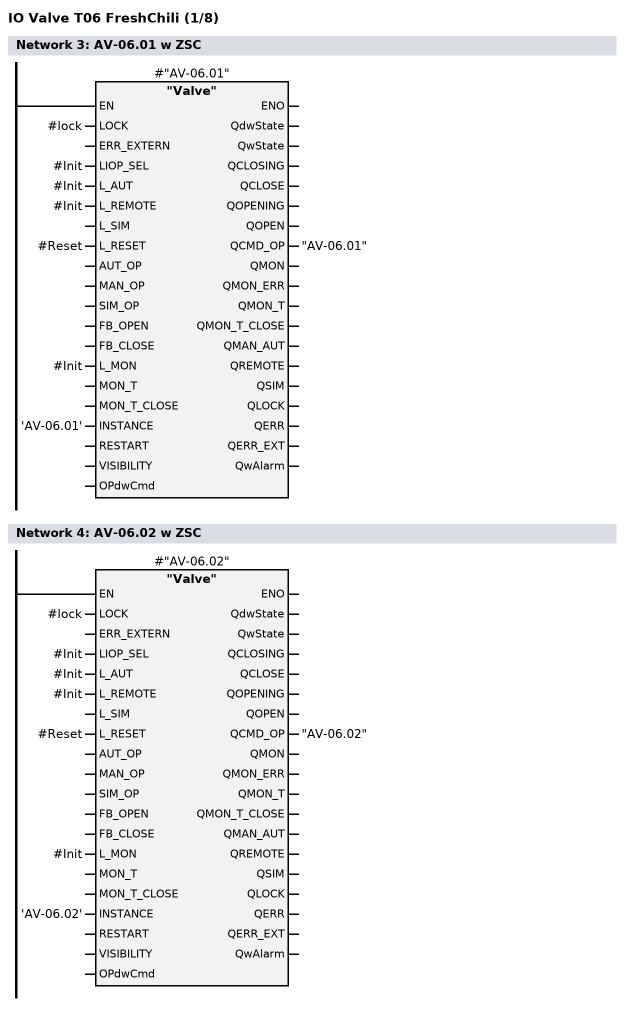
   RUNG wire#powerrail
      #"AV-06.01"(LOCK := #lock, ERR_EXTERN :=, LIOP_SEL := #Init, L_AUT := #Init, L_REMOTE := #Init, L_SIM :=, L_RESET := #Reset, AUT_OP :=, MAN_OP :=, SIM_OP :=, FB_OPEN :=, FB_CLOSE :=, L_MON := #Init, MON_T :=, MON_T_CLOSE :=, INSTANCE := 'AV-06.01', RESTART :=, VISIBILITY :=, OPdwCmd :=, QdwState =>, QwState =>, QCLOSING =>, QCLOSE =>, QOPENING =>, QOPEN =>, QCMD_OP => "AV-06.01", QMON =>, QMON_ERR =>, QMON_T =>, QMON_T_CLOSE =>, QMAN_AUT =>, QREMOTE =>, QSIM =>, QLOCK =>, QERR =>, QERR_EXT =>, QwAlarm =>)
   END_RUNG
   // the same network as SCL:
   #"AV-06.01"(LOCK := #lock,   // "Valve"
               LIOP_SEL := #Init,
               L_AUT := #Init,
               L_REMOTE := #Init,
               L_RESET := #Reset,
               L_MON := #Init,
               INSTANCE := 'AV-06.01',
               QCMD_OP => "AV-06.01");
END_REGION

REGION Network 4: AV-06.02 w ZSC
   RUNG wire#powerrail
      #"AV-06.02"(LOCK := #lock, ERR_EXTERN :=, LIOP_SEL := #Init, L_AUT := #Init, L_REMOTE := #Init, L_SIM :=, L_RESET := #Reset, AUT_OP :=, MAN_OP :=, SIM_OP :=, FB_OPEN :=, FB_CLOSE :=, L_MON := #Init, MON_T :=, MON_T_CLOSE :=, INSTANCE := 'AV-06.02', RESTART :=, VISIBILITY :=, OPdwCmd :=, QdwState =>, QwState =>, QCLOSING =>, QCLOSE =>, QOPENING =>, QOPEN =>, QCMD_OP => "AV-06.02", QMON =>, QMON_ERR =>, QMON_T =>, QMON_T_CLOSE =>, QMAN_AUT =>, QREMOTE =>, QSIM =>, QLOCK =>, QERR =>, QERR_EXT =>, QwAlarm =>)
   END_RUNG
   // the same network as SCL:
   #"AV-06.02"(LOCK := #lock,   // "Valve"
               LIOP_SEL := #Init,
               L_AUT := #Init,
               L_REMOTE := #Init,
               L_RESET := #Reset,
               L_MON := #Init,
               INSTANCE := 'AV-06.02',
               QCMD_OP => "AV-06.02");
END_REGION

REGION Network 5: AV-06.03 w ZSC
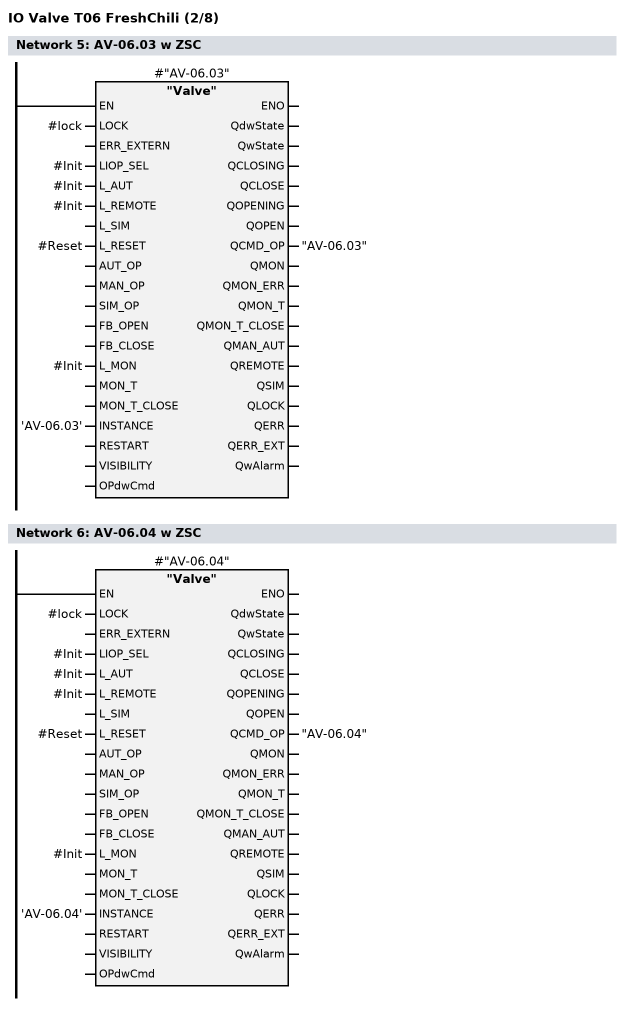
   RUNG wire#powerrail
      #"AV-06.03"(LOCK := #lock, ERR_EXTERN :=, LIOP_SEL := #Init, L_AUT := #Init, L_REMOTE := #Init, L_SIM :=, L_RESET := #Reset, AUT_OP :=, MAN_OP :=, SIM_OP :=, FB_OPEN :=, FB_CLOSE :=, L_MON := #Init, MON_T :=, MON_T_CLOSE :=, INSTANCE := 'AV-06.03', RESTART :=, VISIBILITY :=, OPdwCmd :=, QdwState =>, QwState =>, QCLOSING =>, QCLOSE =>, QOPENING =>, QOPEN =>, QCMD_OP => "AV-06.03", QMON =>, QMON_ERR =>, QMON_T =>, QMON_T_CLOSE =>, QMAN_AUT =>, QREMOTE =>, QSIM =>, QLOCK =>, QERR =>, QERR_EXT =>, QwAlarm =>)
   END_RUNG
   // the same network as SCL:
   #"AV-06.03"(LOCK := #lock,   // "Valve"
               LIOP_SEL := #Init,
               L_AUT := #Init,
               L_REMOTE := #Init,
               L_RESET := #Reset,
               L_MON := #Init,
               INSTANCE := 'AV-06.03',
               QCMD_OP => "AV-06.03");
END_REGION

REGION Network 6: AV-06.04 w ZSC
   RUNG wire#powerrail
      #"AV-06.04"(LOCK := #lock, ERR_EXTERN :=, LIOP_SEL := #Init, L_AUT := #Init, L_REMOTE := #Init, L_SIM :=, L_RESET := #Reset, AUT_OP :=, MAN_OP :=, SIM_OP :=, FB_OPEN :=, FB_CLOSE :=, L_MON := #Init, MON_T :=, MON_T_CLOSE :=, INSTANCE := 'AV-06.04', RESTART :=, VISIBILITY :=, OPdwCmd :=, QdwState =>, QwState =>, QCLOSING =>, QCLOSE =>, QOPENING =>, QOPEN =>, QCMD_OP => "AV-06.04", QMON =>, QMON_ERR =>, QMON_T =>, QMON_T_CLOSE =>, QMAN_AUT =>, QREMOTE =>, QSIM =>, QLOCK =>, QERR =>, QERR_EXT =>, QwAlarm =>)
   END_RUNG
   // the same network as SCL:
   #"AV-06.04"(LOCK := #lock,   // "Valve"
               LIOP_SEL := #Init,
               L_AUT := #Init,
               L_REMOTE := #Init,
               L_RESET := #Reset,
               L_MON := #Init,
               INSTANCE := 'AV-06.04',
               QCMD_OP => "AV-06.04");
END_REGION

REGION Network 7: AV-06.05
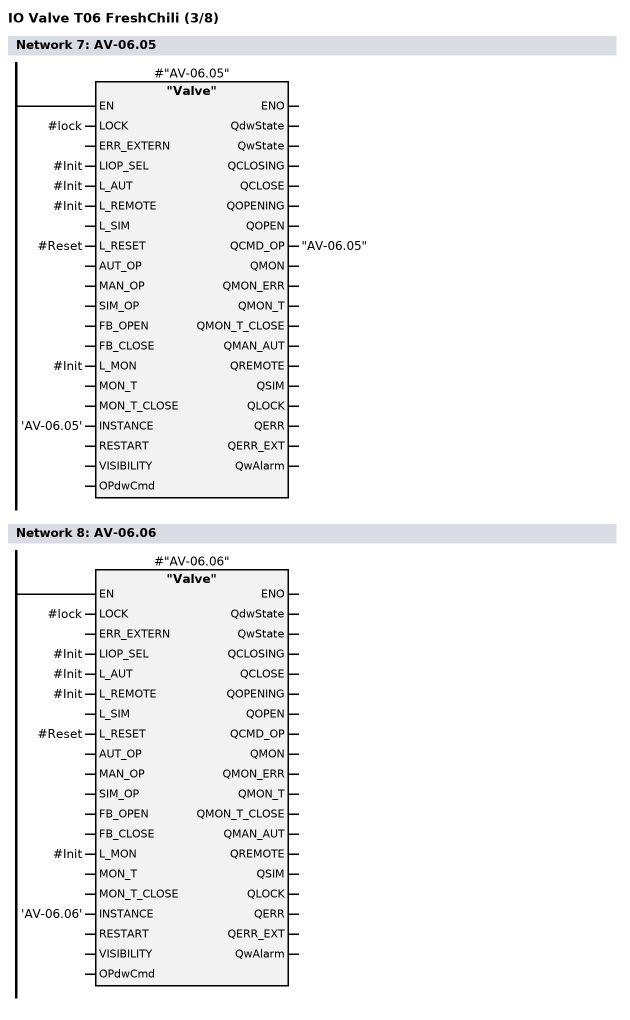
   RUNG wire#powerrail
      #"AV-06.05"(LOCK := #lock, ERR_EXTERN :=, LIOP_SEL := #Init, L_AUT := #Init, L_REMOTE := #Init, L_SIM :=, L_RESET := #Reset, AUT_OP :=, MAN_OP :=, SIM_OP :=, FB_OPEN :=, FB_CLOSE :=, L_MON := #Init, MON_T :=, MON_T_CLOSE :=, INSTANCE := 'AV-06.05', RESTART :=, VISIBILITY :=, OPdwCmd :=, QdwState =>, QwState =>, QCLOSING =>, QCLOSE =>, QOPENING =>, QOPEN =>, QCMD_OP => "AV-06.05", QMON =>, QMON_ERR =>, QMON_T =>, QMON_T_CLOSE =>, QMAN_AUT =>, QREMOTE =>, QSIM =>, QLOCK =>, QERR =>, QERR_EXT =>, QwAlarm =>)
   END_RUNG
   // the same network as SCL:
   #"AV-06.05"(LOCK := #lock,   // "Valve"
               LIOP_SEL := #Init,
               L_AUT := #Init,
               L_REMOTE := #Init,
               L_RESET := #Reset,
               L_MON := #Init,
               INSTANCE := 'AV-06.05',
               QCMD_OP => "AV-06.05");
END_REGION

REGION Network 8: AV-06.06
   RUNG wire#powerrail
      #"AV-06.06"(LOCK := #lock, ERR_EXTERN :=, LIOP_SEL := #Init, L_AUT := #Init, L_REMOTE := #Init, L_SIM :=, L_RESET := #Reset, AUT_OP :=, MAN_OP :=, SIM_OP :=, FB_OPEN :=, FB_CLOSE :=, L_MON := #Init, MON_T :=, MON_T_CLOSE :=, INSTANCE := 'AV-06.06', RESTART :=, VISIBILITY :=, OPdwCmd :=, QdwState =>, QwState =>, QCLOSING =>, QCLOSE =>, QOPENING =>, QOPEN =>, QCMD_OP =>, QMON =>, QMON_ERR =>, QMON_T =>, QMON_T_CLOSE =>, QMAN_AUT =>, QREMOTE =>, QSIM =>, QLOCK =>, QERR =>, QERR_EXT =>, QwAlarm =>)
   END_RUNG
   // the same network as SCL:
   #"AV-06.06"(LOCK := #lock,   // "Valve"
               LIOP_SEL := #Init,
               L_AUT := #Init,
               L_REMOTE := #Init,
               L_RESET := #Reset,
               L_MON := #Init,
               INSTANCE := 'AV-06.06');
END_REGION

REGION Network 9: AV-06.07
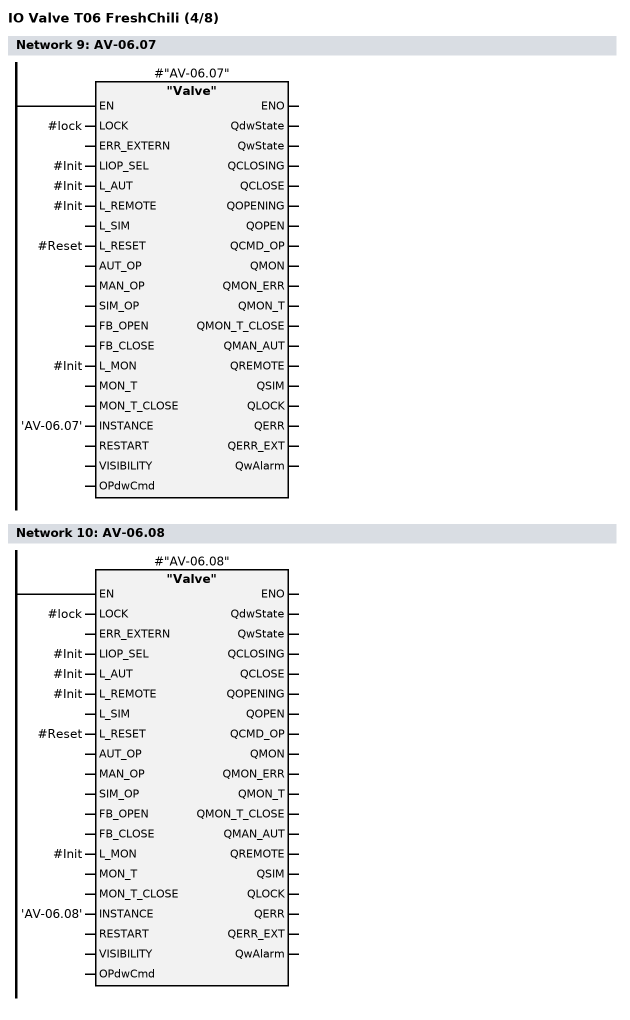
   RUNG wire#powerrail
      #"AV-06.07"(LOCK := #lock, ERR_EXTERN :=, LIOP_SEL := #Init, L_AUT := #Init, L_REMOTE := #Init, L_SIM :=, L_RESET := #Reset, AUT_OP :=, MAN_OP :=, SIM_OP :=, FB_OPEN :=, FB_CLOSE :=, L_MON := #Init, MON_T :=, MON_T_CLOSE :=, INSTANCE := 'AV-06.07', RESTART :=, VISIBILITY :=, OPdwCmd :=, QdwState =>, QwState =>, QCLOSING =>, QCLOSE =>, QOPENING =>, QOPEN =>, QCMD_OP =>, QMON =>, QMON_ERR =>, QMON_T =>, QMON_T_CLOSE =>, QMAN_AUT =>, QREMOTE =>, QSIM =>, QLOCK =>, QERR =>, QERR_EXT =>, QwAlarm =>)
   END_RUNG
   // the same network as SCL:
   #"AV-06.07"(LOCK := #lock,   // "Valve"
               LIOP_SEL := #Init,
               L_AUT := #Init,
               L_REMOTE := #Init,
               L_RESET := #Reset,
               L_MON := #Init,
               INSTANCE := 'AV-06.07');
END_REGION

REGION Network 10: AV-06.08
   RUNG wire#powerrail
      #"AV-06.08"(LOCK := #lock, ERR_EXTERN :=, LIOP_SEL := #Init, L_AUT := #Init, L_REMOTE := #Init, L_SIM :=, L_RESET := #Reset, AUT_OP :=, MAN_OP :=, SIM_OP :=, FB_OPEN :=, FB_CLOSE :=, L_MON := #Init, MON_T :=, MON_T_CLOSE :=, INSTANCE := 'AV-06.08', RESTART :=, VISIBILITY :=, OPdwCmd :=, QdwState =>, QwState =>, QCLOSING =>, QCLOSE =>, QOPENING =>, QOPEN =>, QCMD_OP =>, QMON =>, QMON_ERR =>, QMON_T =>, QMON_T_CLOSE =>, QMAN_AUT =>, QREMOTE =>, QSIM =>, QLOCK =>, QERR =>, QERR_EXT =>, QwAlarm =>)
   END_RUNG
   // the same network as SCL:
   #"AV-06.08"(LOCK := #lock,   // "Valve"
               LIOP_SEL := #Init,
               L_AUT := #Init,
               L_REMOTE := #Init,
               L_RESET := #Reset,
               L_MON := #Init,
               INSTANCE := 'AV-06.08');
END_REGION

REGION Network 11: AV-06.09
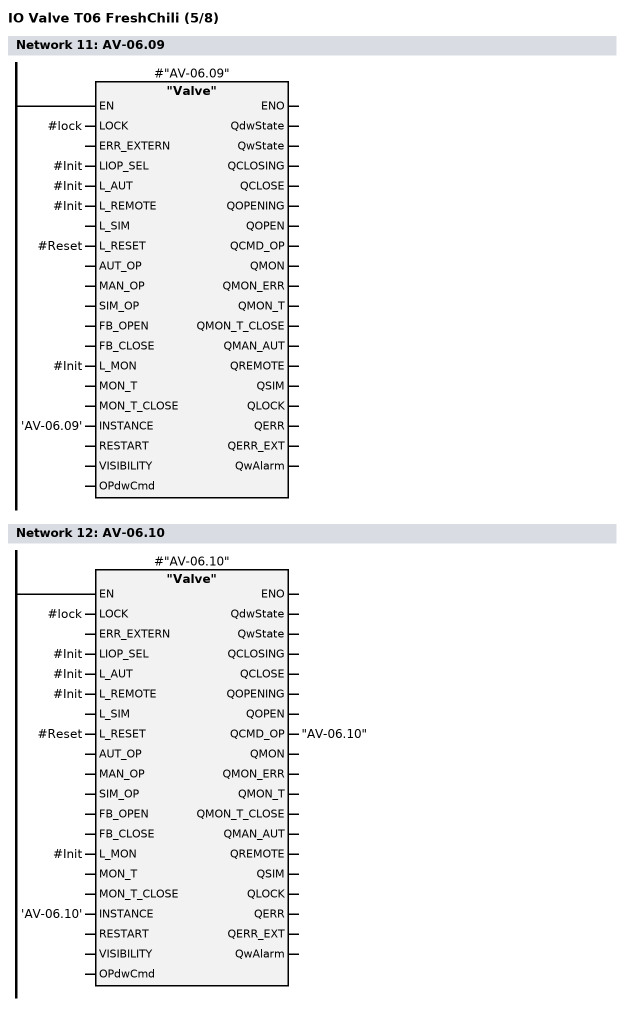
   RUNG wire#powerrail
      #"AV-06.09"(LOCK := #lock, ERR_EXTERN :=, LIOP_SEL := #Init, L_AUT := #Init, L_REMOTE := #Init, L_SIM :=, L_RESET := #Reset, AUT_OP :=, MAN_OP :=, SIM_OP :=, FB_OPEN :=, FB_CLOSE :=, L_MON := #Init, MON_T :=, MON_T_CLOSE :=, INSTANCE := 'AV-06.09', RESTART :=, VISIBILITY :=, OPdwCmd :=, QdwState =>, QwState =>, QCLOSING =>, QCLOSE =>, QOPENING =>, QOPEN =>, QCMD_OP =>, QMON =>, QMON_ERR =>, QMON_T =>, QMON_T_CLOSE =>, QMAN_AUT =>, QREMOTE =>, QSIM =>, QLOCK =>, QERR =>, QERR_EXT =>, QwAlarm =>)
   END_RUNG
   // the same network as SCL:
   #"AV-06.09"(LOCK := #lock,   // "Valve"
               LIOP_SEL := #Init,
               L_AUT := #Init,
               L_REMOTE := #Init,
               L_RESET := #Reset,
               L_MON := #Init,
               INSTANCE := 'AV-06.09');
END_REGION

REGION Network 12: AV-06.10
   RUNG wire#powerrail
      #"AV-06.10"(LOCK := #lock, ERR_EXTERN :=, LIOP_SEL := #Init, L_AUT := #Init, L_REMOTE := #Init, L_SIM :=, L_RESET := #Reset, AUT_OP :=, MAN_OP :=, SIM_OP :=, FB_OPEN :=, FB_CLOSE :=, L_MON := #Init, MON_T :=, MON_T_CLOSE :=, INSTANCE := 'AV-06.10', RESTART :=, VISIBILITY :=, OPdwCmd :=, QdwState =>, QwState =>, QCLOSING =>, QCLOSE =>, QOPENING =>, QOPEN =>, QCMD_OP => "AV-06.10", QMON =>, QMON_ERR =>, QMON_T =>, QMON_T_CLOSE =>, QMAN_AUT =>, QREMOTE =>, QSIM =>, QLOCK =>, QERR =>, QERR_EXT =>, QwAlarm =>)
   END_RUNG
   // the same network as SCL:
   #"AV-06.10"(LOCK := #lock,   // "Valve"
               LIOP_SEL := #Init,
               L_AUT := #Init,
               L_REMOTE := #Init,
               L_RESET := #Reset,
               L_MON := #Init,
               INSTANCE := 'AV-06.10',
               QCMD_OP => "AV-06.10");
END_REGION

REGION Network 13: AV-06.11 w ZSC
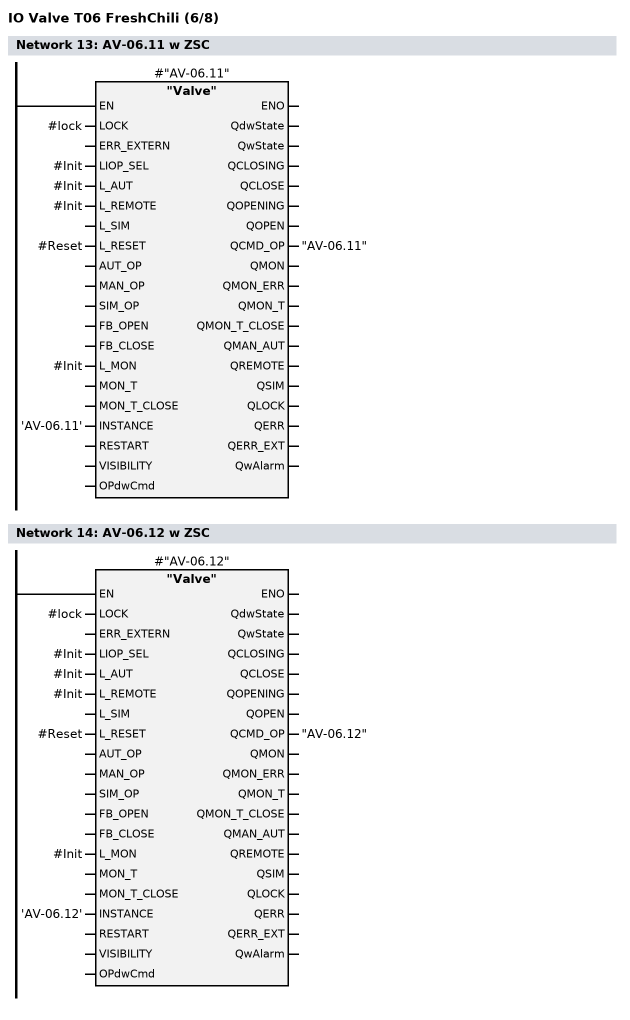
   RUNG wire#powerrail
      #"AV-06.11"(LOCK := #lock, ERR_EXTERN :=, LIOP_SEL := #Init, L_AUT := #Init, L_REMOTE := #Init, L_SIM :=, L_RESET := #Reset, AUT_OP :=, MAN_OP :=, SIM_OP :=, FB_OPEN :=, FB_CLOSE :=, L_MON := #Init, MON_T :=, MON_T_CLOSE :=, INSTANCE := 'AV-06.11', RESTART :=, VISIBILITY :=, OPdwCmd :=, QdwState =>, QwState =>, QCLOSING =>, QCLOSE =>, QOPENING =>, QOPEN =>, QCMD_OP => "AV-06.11", QMON =>, QMON_ERR =>, QMON_T =>, QMON_T_CLOSE =>, QMAN_AUT =>, QREMOTE =>, QSIM =>, QLOCK =>, QERR =>, QERR_EXT =>, QwAlarm =>)
   END_RUNG
   // the same network as SCL:
   #"AV-06.11"(LOCK := #lock,   // "Valve"
               LIOP_SEL := #Init,
               L_AUT := #Init,
               L_REMOTE := #Init,
               L_RESET := #Reset,
               L_MON := #Init,
               INSTANCE := 'AV-06.11',
               QCMD_OP => "AV-06.11");
END_REGION

REGION Network 14: AV-06.12 w ZSC
   RUNG wire#powerrail
      #"AV-06.12"(LOCK := #lock, ERR_EXTERN :=, LIOP_SEL := #Init, L_AUT := #Init, L_REMOTE := #Init, L_SIM :=, L_RESET := #Reset, AUT_OP :=, MAN_OP :=, SIM_OP :=, FB_OPEN :=, FB_CLOSE :=, L_MON := #Init, MON_T :=, MON_T_CLOSE :=, INSTANCE := 'AV-06.12', RESTART :=, VISIBILITY :=, OPdwCmd :=, QdwState =>, QwState =>, QCLOSING =>, QCLOSE =>, QOPENING =>, QOPEN =>, QCMD_OP => "AV-06.12", QMON =>, QMON_ERR =>, QMON_T =>, QMON_T_CLOSE =>, QMAN_AUT =>, QREMOTE =>, QSIM =>, QLOCK =>, QERR =>, QERR_EXT =>, QwAlarm =>)
   END_RUNG
   // the same network as SCL:
   #"AV-06.12"(LOCK := #lock,   // "Valve"
               LIOP_SEL := #Init,
               L_AUT := #Init,
               L_REMOTE := #Init,
               L_RESET := #Reset,
               L_MON := #Init,
               INSTANCE := 'AV-06.12',
               QCMD_OP => "AV-06.12");
END_REGION

REGION Network 15: AV-06.13 w ZSC
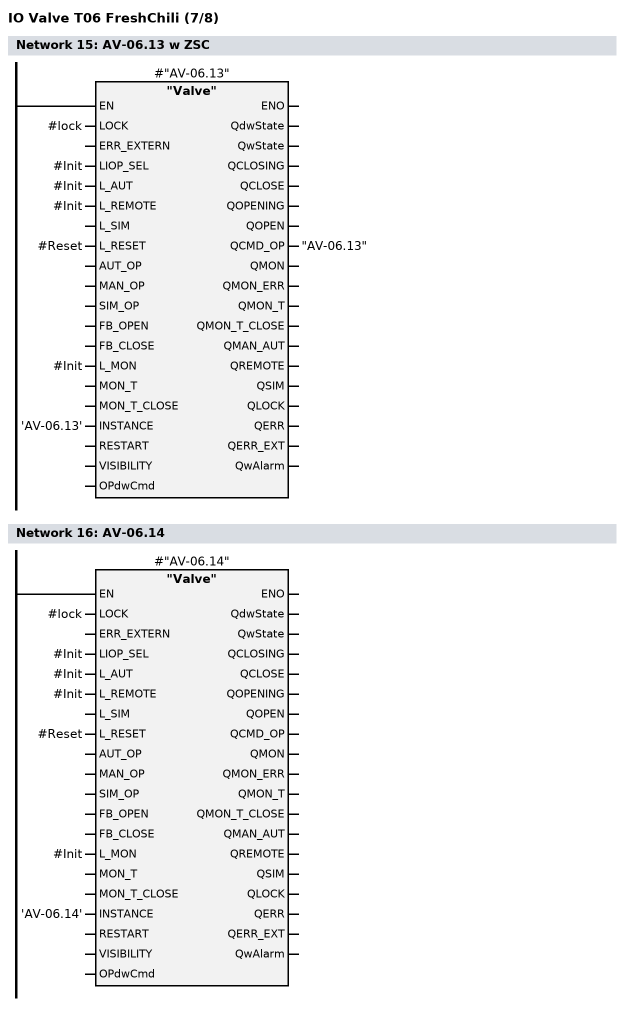
   RUNG wire#powerrail
      #"AV-06.13"(LOCK := #lock, ERR_EXTERN :=, LIOP_SEL := #Init, L_AUT := #Init, L_REMOTE := #Init, L_SIM :=, L_RESET := #Reset, AUT_OP :=, MAN_OP :=, SIM_OP :=, FB_OPEN :=, FB_CLOSE :=, L_MON := #Init, MON_T :=, MON_T_CLOSE :=, INSTANCE := 'AV-06.13', RESTART :=, VISIBILITY :=, OPdwCmd :=, QdwState =>, QwState =>, QCLOSING =>, QCLOSE =>, QOPENING =>, QOPEN =>, QCMD_OP => "AV-06.13", QMON =>, QMON_ERR =>, QMON_T =>, QMON_T_CLOSE =>, QMAN_AUT =>, QREMOTE =>, QSIM =>, QLOCK =>, QERR =>, QERR_EXT =>, QwAlarm =>)
   END_RUNG
   // the same network as SCL:
   #"AV-06.13"(LOCK := #lock,   // "Valve"
               LIOP_SEL := #Init,
               L_AUT := #Init,
               L_REMOTE := #Init,
               L_RESET := #Reset,
               L_MON := #Init,
               INSTANCE := 'AV-06.13',
               QCMD_OP => "AV-06.13");
END_REGION

REGION Network 16: AV-06.14
   RUNG wire#powerrail
      #"AV-06.14"(LOCK := #lock, ERR_EXTERN :=, LIOP_SEL := #Init, L_AUT := #Init, L_REMOTE := #Init, L_SIM :=, L_RESET := #Reset, AUT_OP :=, MAN_OP :=, SIM_OP :=, FB_OPEN :=, FB_CLOSE :=, L_MON := #Init, MON_T :=, MON_T_CLOSE :=, INSTANCE := 'AV-06.14', RESTART :=, VISIBILITY :=, OPdwCmd :=, QdwState =>, QwState =>, QCLOSING =>, QCLOSE =>, QOPENING =>, QOPEN =>, QCMD_OP =>, QMON =>, QMON_ERR =>, QMON_T =>, QMON_T_CLOSE =>, QMAN_AUT =>, QREMOTE =>, QSIM =>, QLOCK =>, QERR =>, QERR_EXT =>, QwAlarm =>)
   END_RUNG
   // the same network as SCL:
   #"AV-06.14"(LOCK := #lock,   // "Valve"
               LIOP_SEL := #Init,
               L_AUT := #Init,
               L_REMOTE := #Init,
               L_RESET := #Reset,
               L_MON := #Init,
               INSTANCE := 'AV-06.14');
END_REGION

REGION Network 17: AV-06.15
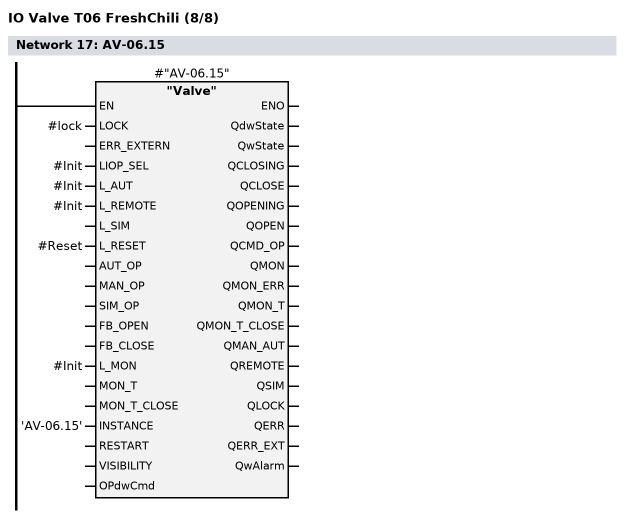
   RUNG wire#powerrail
      #"AV-06.15"(LOCK := #lock, ERR_EXTERN :=, LIOP_SEL := #Init, L_AUT := #Init, L_REMOTE := #Init, L_SIM :=, L_RESET := #Reset, AUT_OP :=, MAN_OP :=, SIM_OP :=, FB_OPEN :=, FB_CLOSE :=, L_MON := #Init, MON_T :=, MON_T_CLOSE :=, INSTANCE := 'AV-06.15', RESTART :=, VISIBILITY :=, OPdwCmd :=, QdwState =>, QwState =>, QCLOSING =>, QCLOSE =>, QOPENING =>, QOPEN =>, QCMD_OP =>, QMON =>, QMON_ERR =>, QMON_T =>, QMON_T_CLOSE =>, QMAN_AUT =>, QREMOTE =>, QSIM =>, QLOCK =>, QERR =>, QERR_EXT =>, QwAlarm =>)
   END_RUNG
   // the same network as SCL:
   #"AV-06.15"(LOCK := #lock,   // "Valve"
               LIOP_SEL := #Init,
               L_AUT := #Init,
               L_REMOTE := #Init,
               L_RESET := #Reset,
               L_MON := #Init,
               INSTANCE := 'AV-06.15');
END_REGION
END_FUNCTION_BLOCK

FUNCTION_BLOCK "IO Valve T07 FreshChili"   // FB307, LAD
{ S7_Optimized_Access := 'FALSE' }
VERSION : 0.1
// stored: AutoNumber false, IsIECCheckEnabled false, SetENOAutomatically false, UDAEnableTagReadback false
   VAR_INPUT
      lock : Bool;
      Init : Bool;
      testing : Bool;
      Reset : Bool;
   END_VAR
   VAR
      "AV-07.01" { S7_SetPoint := 'True'} : "Valve";   // AUTO BUTTERFLY VALVE INLET PROCESS WATER TO BFT CHILI FRESH T-07.00
      "AV-07.02" { S7_SetPoint := 'True'} : "Valve";   // AUTO BUTTERFLY VALVE CIP SUPPLY TO BFT CHILI FRESH T-07.00
      "AV-07.03" { S7_SetPoint := 'True'} : "Valve";   // AUTO BUTTERFLY VALVE OUTLET PRODUCT FROM BFT CHILI FRESH T-07.00
      "AV-07.04" { S7_SetPoint := 'True'} : "Valve";   // AUTO BUTTERFLY VALVE OUTLET CIP TANK & LINE CHILI FRESH T-07.00
      "AV-07.05" { S7_SetPoint := 'True'} : "Valve";   // AUTO BUTTERFLY VALVE DRAIN MONO PUMP P-07.01
      "AV-07.06" { S7_SetPoint := 'True'} : "Valve";   // AUTO BUTTERFLY VALVE INLET PRODUCT FROM REWORK T-22.00 TO BLENDING TANK T-20.00
      "AV-07.07" { S7_SetPoint := 'True'} : "Valve";
      "AV-07.08" { S7_SetPoint := 'True'} : "Valve";
      "AV-07.09" { S7_SetPoint := 'True'} : "Valve";
      "AV-07.10" { S7_SetPoint := 'True'} : "Valve";
      "AV-07.11" { S7_SetPoint := 'True'} : "Valve";
      "AV-07.12" { S7_SetPoint := 'True'} : "Valve";
      "AV-07.13" { S7_SetPoint := 'True'} : "Valve";
      "AV-07.14" { S7_SetPoint := 'True'} : "Valve";
      "AV-07.15" { S7_SetPoint := 'True'} : "Valve";
   END_VAR
BEGIN

REGION Network 1 (SCL): FB OPEN and CLOSE
   IF #testing THEN
       // Statement section IF
       #"AV-07.01".FB_OPEN := #"AV-07.01".QCMD_OP;
       #"AV-07.01".FB_CLOSE := NOT #"AV-07.01".QCMD_OP;
       #"AV-07.02".FB_OPEN := #"AV-07.02".QCMD_OP;
       #"AV-07.02".FB_CLOSE := NOT #"AV-07.02".QCMD_OP;
       #"AV-07.03".FB_OPEN := #"AV-07.03".QCMD_OP;
       #"AV-07.03".FB_CLOSE := NOT #"AV-07.03".QCMD_OP;
       #"AV-07.04".FB_OPEN := #"AV-07.04".QCMD_OP;
       #"AV-07.04".FB_CLOSE := NOT #"AV-07.04".QCMD_OP;
       #"AV-07.05".FB_OPEN := #"AV-07.05".QCMD_OP;
       #"AV-07.05".FB_CLOSE := NOT #"AV-07.05".QCMD_OP;
       #"AV-07.06".FB_OPEN := #"AV-07.06".QCMD_OP;
       #"AV-07.06".FB_CLOSE := NOT #"AV-07.06".QCMD_OP;
       #"AV-07.07".FB_OPEN := #"AV-07.07".QCMD_OP;
       #"AV-07.07".FB_CLOSE := NOT #"AV-07.07".QCMD_OP;
       #"AV-07.08".FB_OPEN := #"AV-07.08".QCMD_OP;
       #"AV-07.08".FB_CLOSE := NOT #"AV-07.08".QCMD_OP;
       #"AV-07.09".FB_OPEN := #"AV-07.09".QCMD_OP;
       #"AV-07.09".FB_CLOSE := NOT #"AV-07.09".QCMD_OP;
       #"AV-07.10".FB_OPEN := #"AV-07.10".QCMD_OP;
       #"AV-07.10".FB_CLOSE := NOT #"AV-07.10".QCMD_OP;
       #"AV-07.11".FB_OPEN := #"AV-07.11".QCMD_OP;
       #"AV-07.11".FB_CLOSE := NOT #"AV-07.11".QCMD_OP;
       #"AV-07.12".FB_OPEN := #"AV-07.12".QCMD_OP;
       #"AV-07.12".FB_CLOSE := NOT #"AV-07.12".QCMD_OP;
       #"AV-07.13".FB_OPEN := #"AV-07.13".QCMD_OP;
       #"AV-07.13".FB_CLOSE := NOT #"AV-07.13".QCMD_OP;
       #"AV-07.14".FB_OPEN := #"AV-07.14".QCMD_OP;
       #"AV-07.14".FB_CLOSE := NOT #"AV-07.14".QCMD_OP;
       #"AV-07.15".FB_OPEN := #"AV-07.15".QCMD_OP;
       #"AV-07.15".FB_CLOSE := NOT #"AV-07.15".QCMD_OP;
   ELSE
       // Statement section ELSE
       #"AV-07.01".FB_OPEN := NOT "ZSC-07.01";
       #"AV-07.01".FB_CLOSE := "ZSC-07.01";
       #"AV-07.02".FB_OPEN := NOT "ZSC-07.02";
       #"AV-07.02".FB_CLOSE := "ZSC-07.02";
       #"AV-07.03".FB_OPEN := NOT "ZSC-07.03";
       #"AV-07.03".FB_CLOSE := "ZSC-07.03";
       #"AV-07.04".FB_OPEN := NOT "ZSC-07.04";
       #"AV-07.04".FB_CLOSE := "ZSC-07.04";
       #"AV-07.05".FB_OPEN := #"AV-07.05".QCMD_OP;
       #"AV-07.05".FB_CLOSE := NOT #"AV-07.05".QCMD_OP;
       #"AV-07.06".FB_OPEN := #"AV-07.06".QCMD_OP;
       #"AV-07.06".FB_CLOSE := NOT #"AV-07.06".QCMD_OP;
       #"AV-07.07".FB_OPEN := #"AV-07.07".QCMD_OP;
       #"AV-07.07".FB_CLOSE := NOT #"AV-07.07".QCMD_OP;
       #"AV-07.08".FB_OPEN := #"AV-07.08".QCMD_OP;
       #"AV-07.08".FB_CLOSE := NOT #"AV-07.08".QCMD_OP;
       #"AV-07.09".FB_OPEN := #"AV-07.09".QCMD_OP;
       #"AV-07.09".FB_CLOSE := NOT #"AV-07.09".QCMD_OP;
       #"AV-07.10".FB_OPEN := #"AV-07.10".QCMD_OP;
       #"AV-07.10".FB_CLOSE := NOT #"AV-07.10".QCMD_OP;
       #"AV-07.11".FB_OPEN := NOT "ZSC-07.11";
       #"AV-07.11".FB_CLOSE := "ZSC-07.11";
       #"AV-07.12".FB_OPEN := NOT "ZSC-07.12";
       #"AV-07.12".FB_CLOSE := "ZSC-07.12";
       #"AV-07.13".FB_OPEN := NOT "ZSC-07.13";
       #"AV-07.13".FB_CLOSE := "ZSC-07.13";
       #"AV-07.14".FB_OPEN := #"AV-07.14".QCMD_OP;
       #"AV-07.14".FB_CLOSE := NOT #"AV-07.14".QCMD_OP;
       #"AV-07.15".FB_OPEN := #"AV-07.15".QCMD_OP;
       #"AV-07.15".FB_CLOSE := NOT #"AV-07.15".QCMD_OP;
   END_IF;
END_REGION

NETWORK
TITLE = FB Monitoring Time
// FB OPEN Time
      L     t#20s;
      T     #"AV-07.01".MON_T;
      T     #"AV-07.02".MON_T;
      T     #"AV-07.03".MON_T;
      T     #"AV-07.04".MON_T;
      T     #"AV-07.05".MON_T;
      T     #"AV-07.06".MON_T;
      T     #"AV-07.07".MON_T;
      T     #"AV-07.08".MON_T;
      T     #"AV-07.09".MON_T;
      T     #"AV-07.10".MON_T;
      T     #"AV-07.11".MON_T;
      T     #"AV-07.12".MON_T;
      T     #"AV-07.13".MON_T;
      T     #"AV-07.14".MON_T;
      T     #"AV-07.15".MON_T;
// FB CLOSE Time
      L     t#20s;
      T     #"AV-07.01".MON_T_CLOSE;
      T     #"AV-07.02".MON_T_CLOSE;
      T     #"AV-07.03".MON_T_CLOSE;
      T     #"AV-07.04".MON_T_CLOSE;
      T     #"AV-07.05".MON_T_CLOSE;
      T     #"AV-07.06".MON_T_CLOSE;
      T     #"AV-07.07".MON_T_CLOSE;
      T     #"AV-07.08".MON_T_CLOSE;
      T     #"AV-07.09".MON_T_CLOSE;
      T     #"AV-07.10".MON_T_CLOSE;
      T     #"AV-07.11".MON_T_CLOSE;
      T     #"AV-07.12".MON_T_CLOSE;
      T     #"AV-07.13".MON_T_CLOSE;
      T     #"AV-07.14".MON_T_CLOSE;
      T     #"AV-07.15".MON_T_CLOSE;

REGION Network 3: AV-07.01 w ZSC
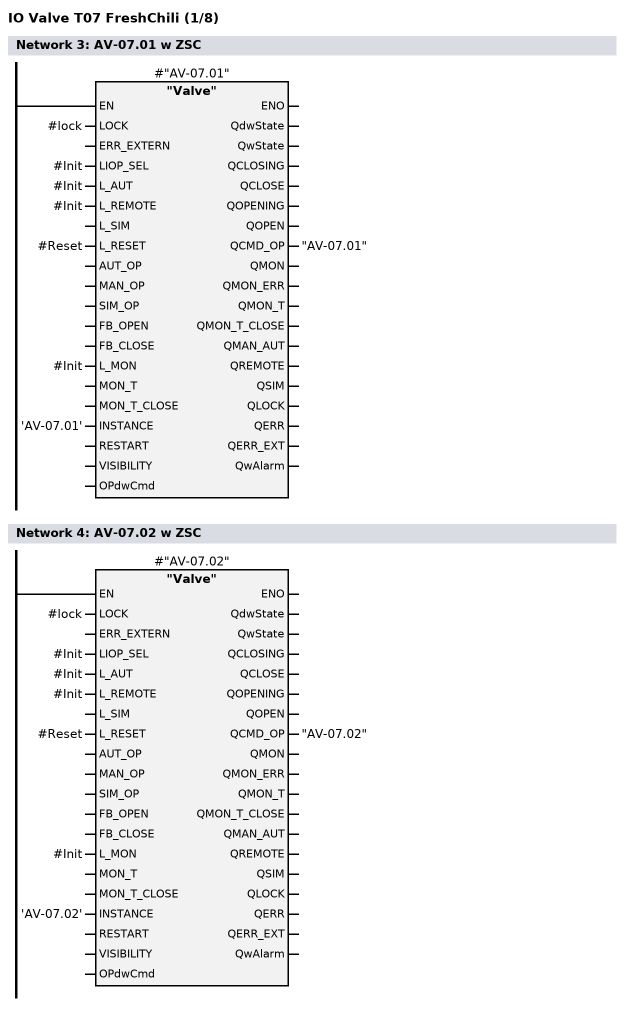
   RUNG wire#powerrail
      #"AV-07.01"(LOCK := #lock, ERR_EXTERN :=, LIOP_SEL := #Init, L_AUT := #Init, L_REMOTE := #Init, L_SIM :=, L_RESET := #Reset, AUT_OP :=, MAN_OP :=, SIM_OP :=, FB_OPEN :=, FB_CLOSE :=, L_MON := #Init, MON_T :=, MON_T_CLOSE :=, INSTANCE := 'AV-07.01', RESTART :=, VISIBILITY :=, OPdwCmd :=, QdwState =>, QwState =>, QCLOSING =>, QCLOSE =>, QOPENING =>, QOPEN =>, QCMD_OP => "AV-07.01", QMON =>, QMON_ERR =>, QMON_T =>, QMON_T_CLOSE =>, QMAN_AUT =>, QREMOTE =>, QSIM =>, QLOCK =>, QERR =>, QERR_EXT =>, QwAlarm =>)
   END_RUNG
   // the same network as SCL:
   #"AV-07.01"(LOCK := #lock,   // "Valve"
               LIOP_SEL := #Init,
               L_AUT := #Init,
               L_REMOTE := #Init,
               L_RESET := #Reset,
               L_MON := #Init,
               INSTANCE := 'AV-07.01',
               QCMD_OP => "AV-07.01");
END_REGION

REGION Network 4: AV-07.02 w ZSC
   RUNG wire#powerrail
      #"AV-07.02"(LOCK := #lock, ERR_EXTERN :=, LIOP_SEL := #Init, L_AUT := #Init, L_REMOTE := #Init, L_SIM :=, L_RESET := #Reset, AUT_OP :=, MAN_OP :=, SIM_OP :=, FB_OPEN :=, FB_CLOSE :=, L_MON := #Init, MON_T :=, MON_T_CLOSE :=, INSTANCE := 'AV-07.02', RESTART :=, VISIBILITY :=, OPdwCmd :=, QdwState =>, QwState =>, QCLOSING =>, QCLOSE =>, QOPENING =>, QOPEN =>, QCMD_OP => "AV-07.02", QMON =>, QMON_ERR =>, QMON_T =>, QMON_T_CLOSE =>, QMAN_AUT =>, QREMOTE =>, QSIM =>, QLOCK =>, QERR =>, QERR_EXT =>, QwAlarm =>)
   END_RUNG
   // the same network as SCL:
   #"AV-07.02"(LOCK := #lock,   // "Valve"
               LIOP_SEL := #Init,
               L_AUT := #Init,
               L_REMOTE := #Init,
               L_RESET := #Reset,
               L_MON := #Init,
               INSTANCE := 'AV-07.02',
               QCMD_OP => "AV-07.02");
END_REGION

REGION Network 5: AV-07.03 w ZSC
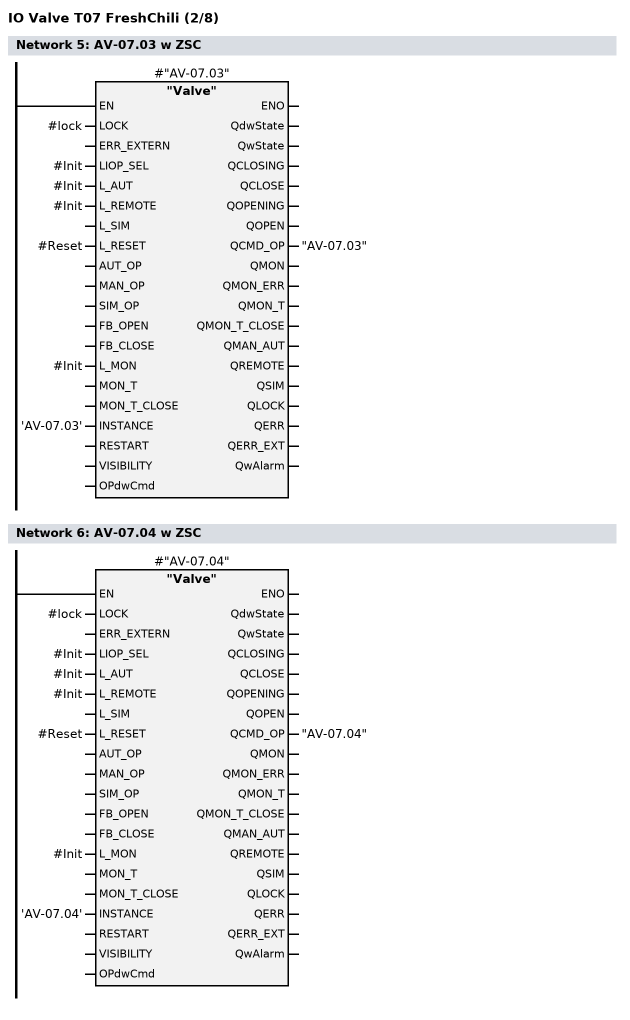
   RUNG wire#powerrail
      #"AV-07.03"(LOCK := #lock, ERR_EXTERN :=, LIOP_SEL := #Init, L_AUT := #Init, L_REMOTE := #Init, L_SIM :=, L_RESET := #Reset, AUT_OP :=, MAN_OP :=, SIM_OP :=, FB_OPEN :=, FB_CLOSE :=, L_MON := #Init, MON_T :=, MON_T_CLOSE :=, INSTANCE := 'AV-07.03', RESTART :=, VISIBILITY :=, OPdwCmd :=, QdwState =>, QwState =>, QCLOSING =>, QCLOSE =>, QOPENING =>, QOPEN =>, QCMD_OP => "AV-07.03", QMON =>, QMON_ERR =>, QMON_T =>, QMON_T_CLOSE =>, QMAN_AUT =>, QREMOTE =>, QSIM =>, QLOCK =>, QERR =>, QERR_EXT =>, QwAlarm =>)
   END_RUNG
   // the same network as SCL:
   #"AV-07.03"(LOCK := #lock,   // "Valve"
               LIOP_SEL := #Init,
               L_AUT := #Init,
               L_REMOTE := #Init,
               L_RESET := #Reset,
               L_MON := #Init,
               INSTANCE := 'AV-07.03',
               QCMD_OP => "AV-07.03");
END_REGION

REGION Network 6: AV-07.04 w ZSC
   RUNG wire#powerrail
      #"AV-07.04"(LOCK := #lock, ERR_EXTERN :=, LIOP_SEL := #Init, L_AUT := #Init, L_REMOTE := #Init, L_SIM :=, L_RESET := #Reset, AUT_OP :=, MAN_OP :=, SIM_OP :=, FB_OPEN :=, FB_CLOSE :=, L_MON := #Init, MON_T :=, MON_T_CLOSE :=, INSTANCE := 'AV-07.04', RESTART :=, VISIBILITY :=, OPdwCmd :=, QdwState =>, QwState =>, QCLOSING =>, QCLOSE =>, QOPENING =>, QOPEN =>, QCMD_OP => "AV-07.04", QMON =>, QMON_ERR =>, QMON_T =>, QMON_T_CLOSE =>, QMAN_AUT =>, QREMOTE =>, QSIM =>, QLOCK =>, QERR =>, QERR_EXT =>, QwAlarm =>)
   END_RUNG
   // the same network as SCL:
   #"AV-07.04"(LOCK := #lock,   // "Valve"
               LIOP_SEL := #Init,
               L_AUT := #Init,
               L_REMOTE := #Init,
               L_RESET := #Reset,
               L_MON := #Init,
               INSTANCE := 'AV-07.04',
               QCMD_OP => "AV-07.04");
END_REGION

REGION Network 7: AV-07.05
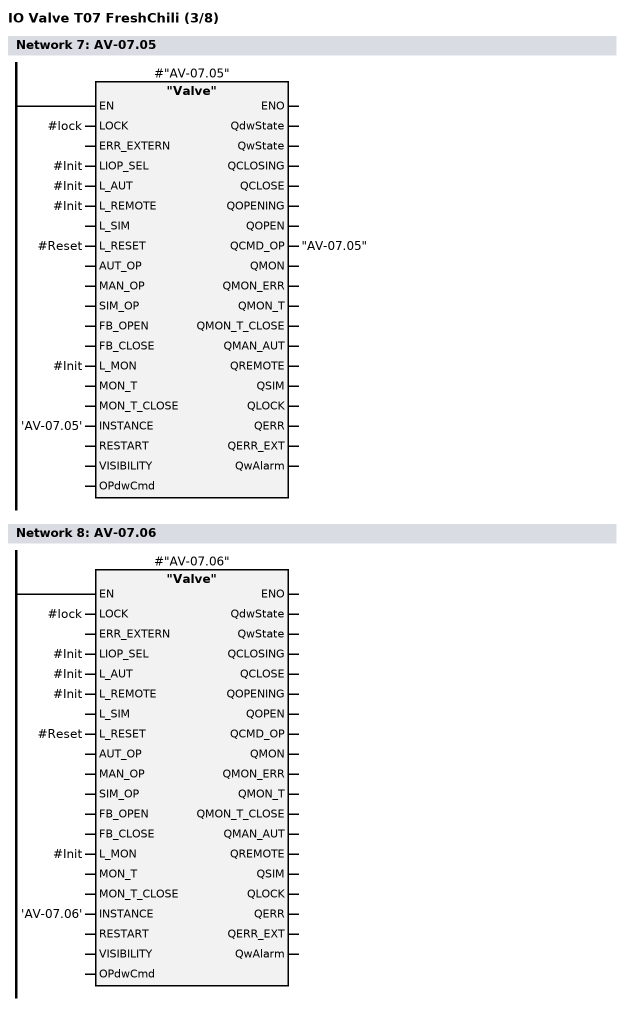
   RUNG wire#powerrail
      #"AV-07.05"(LOCK := #lock, ERR_EXTERN :=, LIOP_SEL := #Init, L_AUT := #Init, L_REMOTE := #Init, L_SIM :=, L_RESET := #Reset, AUT_OP :=, MAN_OP :=, SIM_OP :=, FB_OPEN :=, FB_CLOSE :=, L_MON := #Init, MON_T :=, MON_T_CLOSE :=, INSTANCE := 'AV-07.05', RESTART :=, VISIBILITY :=, OPdwCmd :=, QdwState =>, QwState =>, QCLOSING =>, QCLOSE =>, QOPENING =>, QOPEN =>, QCMD_OP => "AV-07.05", QMON =>, QMON_ERR =>, QMON_T =>, QMON_T_CLOSE =>, QMAN_AUT =>, QREMOTE =>, QSIM =>, QLOCK =>, QERR =>, QERR_EXT =>, QwAlarm =>)
   END_RUNG
   // the same network as SCL:
   #"AV-07.05"(LOCK := #lock,   // "Valve"
               LIOP_SEL := #Init,
               L_AUT := #Init,
               L_REMOTE := #Init,
               L_RESET := #Reset,
               L_MON := #Init,
               INSTANCE := 'AV-07.05',
               QCMD_OP => "AV-07.05");
END_REGION

REGION Network 8: AV-07.06
   RUNG wire#powerrail
      #"AV-07.06"(LOCK := #lock, ERR_EXTERN :=, LIOP_SEL := #Init, L_AUT := #Init, L_REMOTE := #Init, L_SIM :=, L_RESET := #Reset, AUT_OP :=, MAN_OP :=, SIM_OP :=, FB_OPEN :=, FB_CLOSE :=, L_MON := #Init, MON_T :=, MON_T_CLOSE :=, INSTANCE := 'AV-07.06', RESTART :=, VISIBILITY :=, OPdwCmd :=, QdwState =>, QwState =>, QCLOSING =>, QCLOSE =>, QOPENING =>, QOPEN =>, QCMD_OP =>, QMON =>, QMON_ERR =>, QMON_T =>, QMON_T_CLOSE =>, QMAN_AUT =>, QREMOTE =>, QSIM =>, QLOCK =>, QERR =>, QERR_EXT =>, QwAlarm =>)
   END_RUNG
   // the same network as SCL:
   #"AV-07.06"(LOCK := #lock,   // "Valve"
               LIOP_SEL := #Init,
               L_AUT := #Init,
               L_REMOTE := #Init,
               L_RESET := #Reset,
               L_MON := #Init,
               INSTANCE := 'AV-07.06');
END_REGION

REGION Network 9: AV-07.07
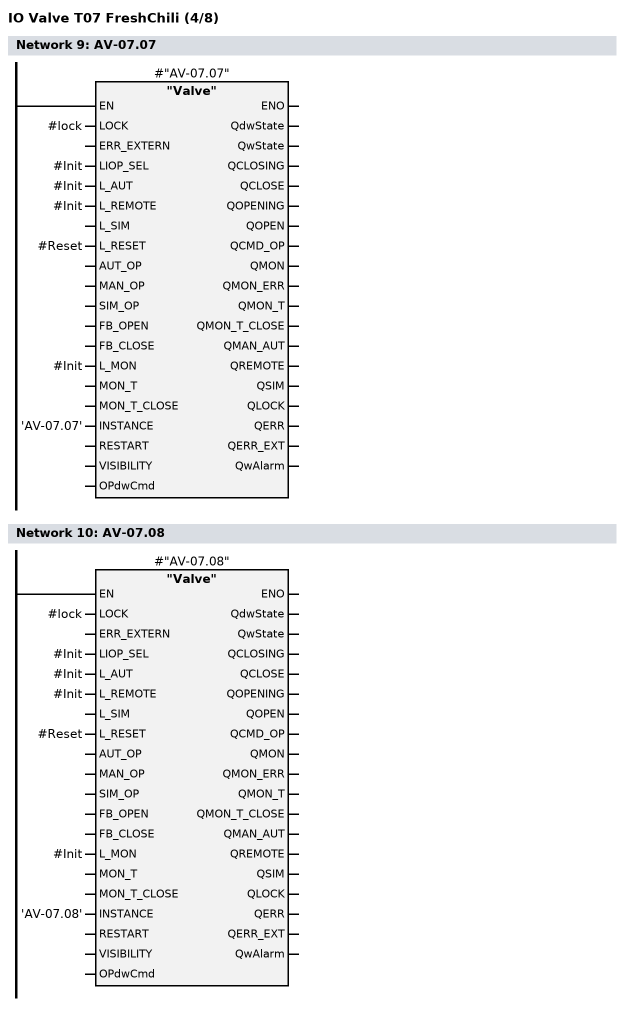
   RUNG wire#powerrail
      #"AV-07.07"(LOCK := #lock, ERR_EXTERN :=, LIOP_SEL := #Init, L_AUT := #Init, L_REMOTE := #Init, L_SIM :=, L_RESET := #Reset, AUT_OP :=, MAN_OP :=, SIM_OP :=, FB_OPEN :=, FB_CLOSE :=, L_MON := #Init, MON_T :=, MON_T_CLOSE :=, INSTANCE := 'AV-07.07', RESTART :=, VISIBILITY :=, OPdwCmd :=, QdwState =>, QwState =>, QCLOSING =>, QCLOSE =>, QOPENING =>, QOPEN =>, QCMD_OP =>, QMON =>, QMON_ERR =>, QMON_T =>, QMON_T_CLOSE =>, QMAN_AUT =>, QREMOTE =>, QSIM =>, QLOCK =>, QERR =>, QERR_EXT =>, QwAlarm =>)
   END_RUNG
   // the same network as SCL:
   #"AV-07.07"(LOCK := #lock,   // "Valve"
               LIOP_SEL := #Init,
               L_AUT := #Init,
               L_REMOTE := #Init,
               L_RESET := #Reset,
               L_MON := #Init,
               INSTANCE := 'AV-07.07');
END_REGION

REGION Network 10: AV-07.08
   RUNG wire#powerrail
      #"AV-07.08"(LOCK := #lock, ERR_EXTERN :=, LIOP_SEL := #Init, L_AUT := #Init, L_REMOTE := #Init, L_SIM :=, L_RESET := #Reset, AUT_OP :=, MAN_OP :=, SIM_OP :=, FB_OPEN :=, FB_CLOSE :=, L_MON := #Init, MON_T :=, MON_T_CLOSE :=, INSTANCE := 'AV-07.08', RESTART :=, VISIBILITY :=, OPdwCmd :=, QdwState =>, QwState =>, QCLOSING =>, QCLOSE =>, QOPENING =>, QOPEN =>, QCMD_OP =>, QMON =>, QMON_ERR =>, QMON_T =>, QMON_T_CLOSE =>, QMAN_AUT =>, QREMOTE =>, QSIM =>, QLOCK =>, QERR =>, QERR_EXT =>, QwAlarm =>)
   END_RUNG
   // the same network as SCL:
   #"AV-07.08"(LOCK := #lock,   // "Valve"
               LIOP_SEL := #Init,
               L_AUT := #Init,
               L_REMOTE := #Init,
               L_RESET := #Reset,
               L_MON := #Init,
               INSTANCE := 'AV-07.08');
END_REGION

REGION Network 11: AV-07.09
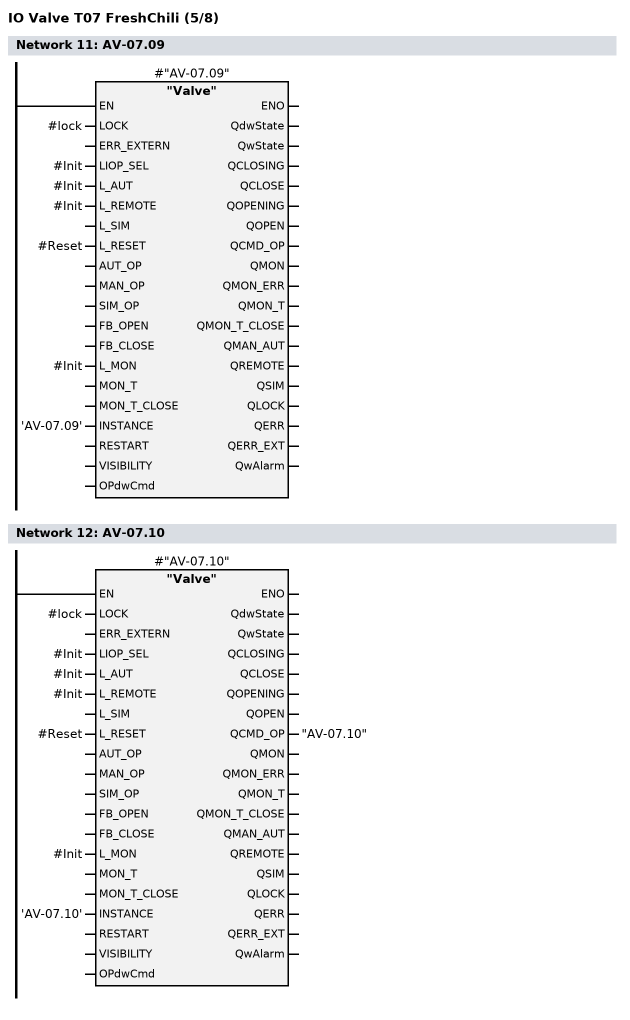
   RUNG wire#powerrail
      #"AV-07.09"(LOCK := #lock, ERR_EXTERN :=, LIOP_SEL := #Init, L_AUT := #Init, L_REMOTE := #Init, L_SIM :=, L_RESET := #Reset, AUT_OP :=, MAN_OP :=, SIM_OP :=, FB_OPEN :=, FB_CLOSE :=, L_MON := #Init, MON_T :=, MON_T_CLOSE :=, INSTANCE := 'AV-07.09', RESTART :=, VISIBILITY :=, OPdwCmd :=, QdwState =>, QwState =>, QCLOSING =>, QCLOSE =>, QOPENING =>, QOPEN =>, QCMD_OP =>, QMON =>, QMON_ERR =>, QMON_T =>, QMON_T_CLOSE =>, QMAN_AUT =>, QREMOTE =>, QSIM =>, QLOCK =>, QERR =>, QERR_EXT =>, QwAlarm =>)
   END_RUNG
   // the same network as SCL:
   #"AV-07.09"(LOCK := #lock,   // "Valve"
               LIOP_SEL := #Init,
               L_AUT := #Init,
               L_REMOTE := #Init,
               L_RESET := #Reset,
               L_MON := #Init,
               INSTANCE := 'AV-07.09');
END_REGION

REGION Network 12: AV-07.10
   RUNG wire#powerrail
      #"AV-07.10"(LOCK := #lock, ERR_EXTERN :=, LIOP_SEL := #Init, L_AUT := #Init, L_REMOTE := #Init, L_SIM :=, L_RESET := #Reset, AUT_OP :=, MAN_OP :=, SIM_OP :=, FB_OPEN :=, FB_CLOSE :=, L_MON := #Init, MON_T :=, MON_T_CLOSE :=, INSTANCE := 'AV-07.10', RESTART :=, VISIBILITY :=, OPdwCmd :=, QdwState =>, QwState =>, QCLOSING =>, QCLOSE =>, QOPENING =>, QOPEN =>, QCMD_OP => "AV-07.10", QMON =>, QMON_ERR =>, QMON_T =>, QMON_T_CLOSE =>, QMAN_AUT =>, QREMOTE =>, QSIM =>, QLOCK =>, QERR =>, QERR_EXT =>, QwAlarm =>)
   END_RUNG
   // the same network as SCL:
   #"AV-07.10"(LOCK := #lock,   // "Valve"
               LIOP_SEL := #Init,
               L_AUT := #Init,
               L_REMOTE := #Init,
               L_RESET := #Reset,
               L_MON := #Init,
               INSTANCE := 'AV-07.10',
               QCMD_OP => "AV-07.10");
END_REGION

REGION Network 13: AV-07.11 w ZSC
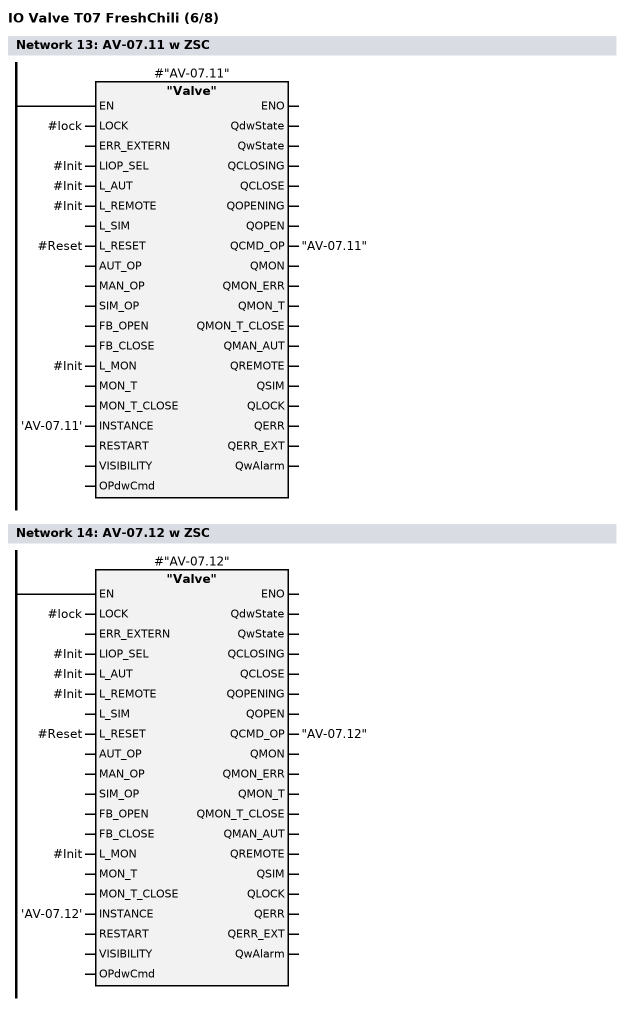
   RUNG wire#powerrail
      #"AV-07.11"(LOCK := #lock, ERR_EXTERN :=, LIOP_SEL := #Init, L_AUT := #Init, L_REMOTE := #Init, L_SIM :=, L_RESET := #Reset, AUT_OP :=, MAN_OP :=, SIM_OP :=, FB_OPEN :=, FB_CLOSE :=, L_MON := #Init, MON_T :=, MON_T_CLOSE :=, INSTANCE := 'AV-07.11', RESTART :=, VISIBILITY :=, OPdwCmd :=, QdwState =>, QwState =>, QCLOSING =>, QCLOSE =>, QOPENING =>, QOPEN =>, QCMD_OP => "AV-07.11", QMON =>, QMON_ERR =>, QMON_T =>, QMON_T_CLOSE =>, QMAN_AUT =>, QREMOTE =>, QSIM =>, QLOCK =>, QERR =>, QERR_EXT =>, QwAlarm =>)
   END_RUNG
   // the same network as SCL:
   #"AV-07.11"(LOCK := #lock,   // "Valve"
               LIOP_SEL := #Init,
               L_AUT := #Init,
               L_REMOTE := #Init,
               L_RESET := #Reset,
               L_MON := #Init,
               INSTANCE := 'AV-07.11',
               QCMD_OP => "AV-07.11");
END_REGION

REGION Network 14: AV-07.12 w ZSC
   RUNG wire#powerrail
      #"AV-07.12"(LOCK := #lock, ERR_EXTERN :=, LIOP_SEL := #Init, L_AUT := #Init, L_REMOTE := #Init, L_SIM :=, L_RESET := #Reset, AUT_OP :=, MAN_OP :=, SIM_OP :=, FB_OPEN :=, FB_CLOSE :=, L_MON := #Init, MON_T :=, MON_T_CLOSE :=, INSTANCE := 'AV-07.12', RESTART :=, VISIBILITY :=, OPdwCmd :=, QdwState =>, QwState =>, QCLOSING =>, QCLOSE =>, QOPENING =>, QOPEN =>, QCMD_OP => "AV-07.12", QMON =>, QMON_ERR =>, QMON_T =>, QMON_T_CLOSE =>, QMAN_AUT =>, QREMOTE =>, QSIM =>, QLOCK =>, QERR =>, QERR_EXT =>, QwAlarm =>)
   END_RUNG
   // the same network as SCL:
   #"AV-07.12"(LOCK := #lock,   // "Valve"
               LIOP_SEL := #Init,
               L_AUT := #Init,
               L_REMOTE := #Init,
               L_RESET := #Reset,
               L_MON := #Init,
               INSTANCE := 'AV-07.12',
               QCMD_OP => "AV-07.12");
END_REGION

REGION Network 15: AV-07.13 w ZSC
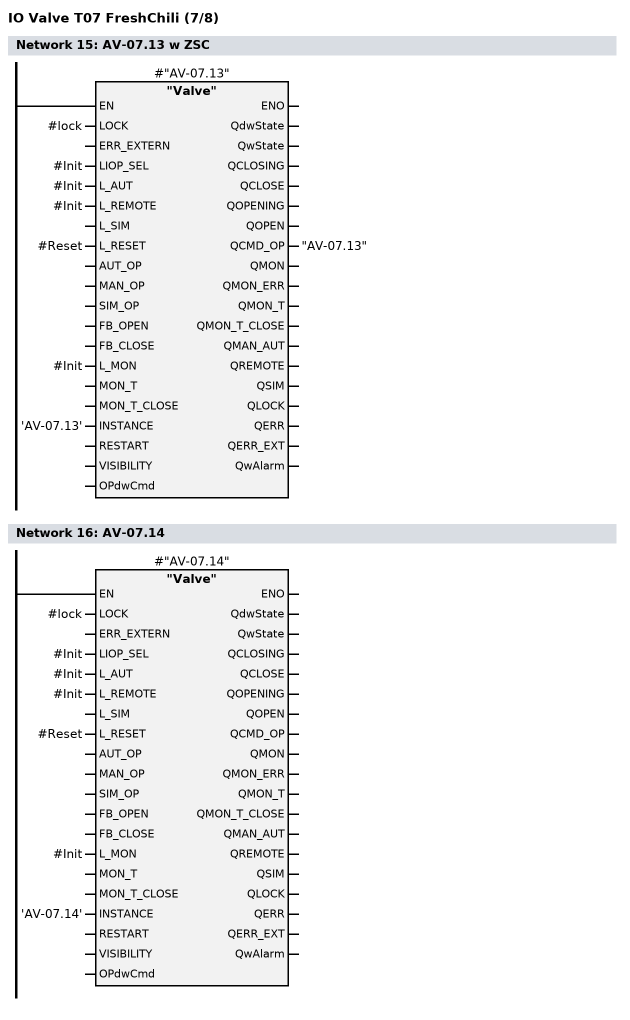
   RUNG wire#powerrail
      #"AV-07.13"(LOCK := #lock, ERR_EXTERN :=, LIOP_SEL := #Init, L_AUT := #Init, L_REMOTE := #Init, L_SIM :=, L_RESET := #Reset, AUT_OP :=, MAN_OP :=, SIM_OP :=, FB_OPEN :=, FB_CLOSE :=, L_MON := #Init, MON_T :=, MON_T_CLOSE :=, INSTANCE := 'AV-07.13', RESTART :=, VISIBILITY :=, OPdwCmd :=, QdwState =>, QwState =>, QCLOSING =>, QCLOSE =>, QOPENING =>, QOPEN =>, QCMD_OP => "AV-07.13", QMON =>, QMON_ERR =>, QMON_T =>, QMON_T_CLOSE =>, QMAN_AUT =>, QREMOTE =>, QSIM =>, QLOCK =>, QERR =>, QERR_EXT =>, QwAlarm =>)
   END_RUNG
   // the same network as SCL:
   #"AV-07.13"(LOCK := #lock,   // "Valve"
               LIOP_SEL := #Init,
               L_AUT := #Init,
               L_REMOTE := #Init,
               L_RESET := #Reset,
               L_MON := #Init,
               INSTANCE := 'AV-07.13',
               QCMD_OP => "AV-07.13");
END_REGION

REGION Network 16: AV-07.14
   RUNG wire#powerrail
      #"AV-07.14"(LOCK := #lock, ERR_EXTERN :=, LIOP_SEL := #Init, L_AUT := #Init, L_REMOTE := #Init, L_SIM :=, L_RESET := #Reset, AUT_OP :=, MAN_OP :=, SIM_OP :=, FB_OPEN :=, FB_CLOSE :=, L_MON := #Init, MON_T :=, MON_T_CLOSE :=, INSTANCE := 'AV-07.14', RESTART :=, VISIBILITY :=, OPdwCmd :=, QdwState =>, QwState =>, QCLOSING =>, QCLOSE =>, QOPENING =>, QOPEN =>, QCMD_OP =>, QMON =>, QMON_ERR =>, QMON_T =>, QMON_T_CLOSE =>, QMAN_AUT =>, QREMOTE =>, QSIM =>, QLOCK =>, QERR =>, QERR_EXT =>, QwAlarm =>)
   END_RUNG
   // the same network as SCL:
   #"AV-07.14"(LOCK := #lock,   // "Valve"
               LIOP_SEL := #Init,
               L_AUT := #Init,
               L_REMOTE := #Init,
               L_RESET := #Reset,
               L_MON := #Init,
               INSTANCE := 'AV-07.14');
END_REGION

REGION Network 17: AV-07.15
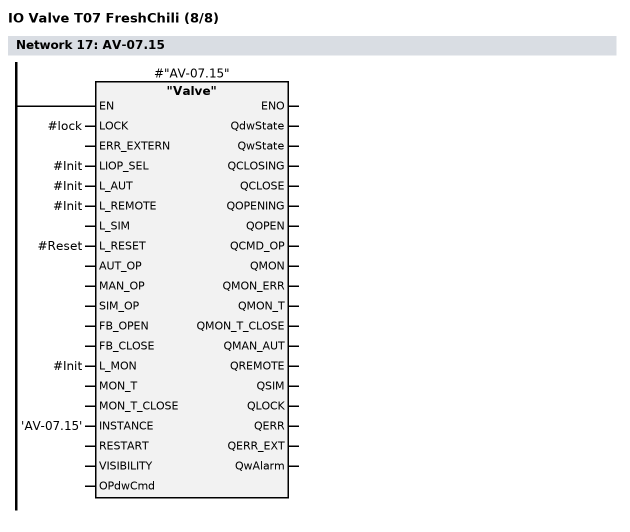
   RUNG wire#powerrail
      #"AV-07.15"(LOCK := #lock, ERR_EXTERN :=, LIOP_SEL := #Init, L_AUT := #Init, L_REMOTE := #Init, L_SIM :=, L_RESET := #Reset, AUT_OP :=, MAN_OP :=, SIM_OP :=, FB_OPEN :=, FB_CLOSE :=, L_MON := #Init, MON_T :=, MON_T_CLOSE :=, INSTANCE := 'AV-07.15', RESTART :=, VISIBILITY :=, OPdwCmd :=, QdwState =>, QwState =>, QCLOSING =>, QCLOSE =>, QOPENING =>, QOPEN =>, QCMD_OP =>, QMON =>, QMON_ERR =>, QMON_T =>, QMON_T_CLOSE =>, QMAN_AUT =>, QREMOTE =>, QSIM =>, QLOCK =>, QERR =>, QERR_EXT =>, QwAlarm =>)
   END_RUNG
   // the same network as SCL:
   #"AV-07.15"(LOCK := #lock,   // "Valve"
               LIOP_SEL := #Init,
               L_AUT := #Init,
               L_REMOTE := #Init,
               L_RESET := #Reset,
               L_MON := #Init,
               INSTANCE := 'AV-07.15');
END_REGION
END_FUNCTION_BLOCK

FUNCTION_BLOCK "IO Valve T08 FreshChili"   // FB308, LAD
{ S7_Optimized_Access := 'FALSE' }
VERSION : 0.1
// stored: AutoNumber false, IsIECCheckEnabled false, SetENOAutomatically false, UDAEnableTagReadback false
   VAR_INPUT
      lock : Bool;
      Init : Bool;
      testing : Bool;
      Reset : Bool;
   END_VAR
   VAR
      "AV-08.01" { S7_SetPoint := 'True'} : "Valve";   // AUTO BUTTERFLY VALVE INLET PROCESS WATER TO BFT CHILI FRESH T-08.00
      "AV-08.02" { S7_SetPoint := 'True'} : "Valve";   // AUTO BUTTERFLY VALVE CIP SUPPLY TO BFT CHILI FRESH T-08.00
      "AV-08.03" { S7_SetPoint := 'True'} : "Valve";   // AUTO BUTTERFLY VALVE OUTLET PRODUCT FROM BFT CHILI FRESH T-08.00
      "AV-08.04" { S7_SetPoint := 'True'} : "Valve";   // AUTO BUTTERFLY VALVE OUTLET CIP TANK & LINE CHILI FRESH T-08.00
      "AV-08.05" { S7_SetPoint := 'True'} : "Valve";   // AUTO BUTTERFLY VALVE DRAIN MONO PUMP P-08.01
      "AV-08.06" { S7_SetPoint := 'True'} : "Valve";   // AUTO BUTTERFLY VALVE INLET PRODUCT FROM REWORK T-22.00 TO BLENDING TANK T-20.00
      "AV-08.07" { S7_SetPoint := 'True'} : "Valve";
      "AV-08.08" { S7_SetPoint := 'True'} : "Valve";
      "AV-08.09" { S7_SetPoint := 'True'} : "Valve";
      "AV-08.10" { S7_SetPoint := 'True'} : "Valve";
      "AV-08.11" { S7_SetPoint := 'True'} : "Valve";
      "AV-08.12" { S7_SetPoint := 'True'} : "Valve";
      "AV-08.13" { S7_SetPoint := 'True'} : "Valve";
      "AV-08.14" { S7_SetPoint := 'True'} : "Valve";
      "AV-08.15" { S7_SetPoint := 'True'} : "Valve";
      "AV-08.16" { S7_SetPoint := 'True'} : "Valve";
      "AV-08.17" { S7_SetPoint := 'True'} : "Valve";
   END_VAR
BEGIN

REGION Network 1 (SCL): FB OPEN and CLOSE
   IF #testing THEN
       // Statement section IF
       #"AV-08.01".FB_OPEN := #"AV-08.01".QCMD_OP;
       #"AV-08.01".FB_CLOSE := NOT #"AV-08.01".QCMD_OP;
       #"AV-08.02".FB_OPEN := #"AV-08.02".QCMD_OP;
       #"AV-08.02".FB_CLOSE := NOT #"AV-08.02".QCMD_OP;
       #"AV-08.03".FB_OPEN := #"AV-08.03".QCMD_OP;
       #"AV-08.03".FB_CLOSE := NOT #"AV-08.03".QCMD_OP;
       #"AV-08.04".FB_OPEN := #"AV-08.04".QCMD_OP;
       #"AV-08.04".FB_CLOSE := NOT #"AV-08.04".QCMD_OP;
       #"AV-08.05".FB_OPEN := #"AV-08.05".QCMD_OP;
       #"AV-08.05".FB_CLOSE := NOT #"AV-08.05".QCMD_OP;
       #"AV-08.06".FB_OPEN := #"AV-08.06".QCMD_OP;
       #"AV-08.06".FB_CLOSE := NOT #"AV-08.06".QCMD_OP;
       #"AV-08.07".FB_OPEN := #"AV-08.07".QCMD_OP;
       #"AV-08.07".FB_CLOSE := NOT #"AV-08.07".QCMD_OP;
       #"AV-08.08".FB_OPEN := #"AV-08.08".QCMD_OP;
       #"AV-08.08".FB_CLOSE := NOT #"AV-08.08".QCMD_OP;
       #"AV-08.09".FB_OPEN := #"AV-08.09".QCMD_OP;
       #"AV-08.09".FB_CLOSE := NOT #"AV-08.09".QCMD_OP;
       #"AV-08.10".FB_OPEN := #"AV-08.10".QCMD_OP;
       #"AV-08.10".FB_CLOSE := NOT #"AV-08.10".QCMD_OP;
       #"AV-08.11".FB_OPEN := #"AV-08.11".QCMD_OP;
       #"AV-08.11".FB_CLOSE := NOT #"AV-08.11".QCMD_OP;
       #"AV-08.12".FB_OPEN := #"AV-08.12".QCMD_OP;
       #"AV-08.12".FB_CLOSE := NOT #"AV-08.12".QCMD_OP;
       #"AV-08.13".FB_OPEN := #"AV-08.13".QCMD_OP;
       #"AV-08.13".FB_CLOSE := NOT #"AV-08.13".QCMD_OP;
       #"AV-08.14".FB_OPEN := #"AV-08.14".QCMD_OP;
       #"AV-08.14".FB_CLOSE := NOT #"AV-08.14".QCMD_OP;
       #"AV-08.15".FB_OPEN := #"AV-08.15".QCMD_OP;
       #"AV-08.15".FB_CLOSE := NOT #"AV-08.15".QCMD_OP;
       #"AV-08.16".FB_OPEN := #"AV-08.16".QCMD_OP;
       #"AV-08.16".FB_CLOSE := NOT #"AV-08.16".QCMD_OP;
       #"AV-08.17".FB_OPEN := #"AV-08.17".QCMD_OP;
       #"AV-08.17".FB_CLOSE := NOT #"AV-08.17".QCMD_OP;
   ELSE
       // Statement section ELSE
       #"AV-08.01".FB_OPEN := NOT "ZSC-08.01";
       #"AV-08.01".FB_CLOSE := "ZSC-08.01";
       #"AV-08.02".FB_OPEN := NOT "ZSC-08.02";
       #"AV-08.02".FB_CLOSE := "ZSC-08.02";
       #"AV-08.03".FB_OPEN := NOT "ZSC-08.03";
       #"AV-08.03".FB_CLOSE := "ZSC-08.03";
       #"AV-08.04".FB_OPEN := NOT "ZSC-08.04";
       #"AV-08.04".FB_CLOSE := "ZSC-08.04";
       #"AV-08.05".FB_OPEN := #"AV-08.05".QCMD_OP;
       #"AV-08.05".FB_CLOSE := NOT #"AV-08.05".QCMD_OP;
       #"AV-08.06".FB_OPEN := #"AV-08.06".QCMD_OP;
       #"AV-08.06".FB_CLOSE := NOT #"AV-08.06".QCMD_OP;
       #"AV-08.07".FB_OPEN := #"AV-08.07".QCMD_OP;
       #"AV-08.07".FB_CLOSE := NOT #"AV-08.07".QCMD_OP;
       #"AV-08.08".FB_OPEN := #"AV-08.08".QCMD_OP;
       #"AV-08.08".FB_CLOSE := NOT #"AV-08.08".QCMD_OP;
       #"AV-08.09".FB_OPEN := #"AV-08.09".QCMD_OP;
       #"AV-08.09".FB_CLOSE := NOT #"AV-08.09".QCMD_OP;
       #"AV-08.10".FB_OPEN := #"AV-08.10".QCMD_OP;
       #"AV-08.10".FB_CLOSE := NOT #"AV-08.10".QCMD_OP;
       #"AV-08.11".FB_OPEN := NOT "ZSC-08.11";
       #"AV-08.11".FB_CLOSE := "ZSC-08.11";
       #"AV-08.12".FB_OPEN := NOT "ZSC-08.12";
       #"AV-08.12".FB_CLOSE := "ZSC-08.12";
       #"AV-08.13".FB_OPEN := NOT "ZSC-08.13";
       #"AV-08.13".FB_CLOSE := "ZSC-08.13";
       #"AV-08.14".FB_OPEN := NOT "ZSC-08.14";
       #"AV-08.14".FB_CLOSE := "ZSC-08.14";
       #"AV-08.15".FB_OPEN := NOT "ZSC-08.15";
       #"AV-08.15".FB_CLOSE := "ZSC-08.15";
       #"AV-08.16".FB_OPEN := #"AV-08.16".QCMD_OP;
       #"AV-08.16".FB_CLOSE := NOT #"AV-08.16".QCMD_OP;
       #"AV-08.17".FB_OPEN := #"AV-08.17".QCMD_OP;
       #"AV-08.17".FB_CLOSE := NOT #"AV-08.17".QCMD_OP;
   END_IF;
END_REGION

NETWORK
TITLE = FB Monitoring Time
// FB OPEN Time
      L     t#20s;
      T     #"AV-08.01".MON_T;
      T     #"AV-08.02".MON_T;
      T     #"AV-08.03".MON_T;
      T     #"AV-08.04".MON_T;
      T     #"AV-08.05".MON_T;
      T     #"AV-08.06".MON_T;
      T     #"AV-08.07".MON_T;
      T     #"AV-08.08".MON_T;
      T     #"AV-08.09".MON_T;
      T     #"AV-08.10".MON_T;
      T     #"AV-08.11".MON_T;
      T     #"AV-08.12".MON_T;
      T     #"AV-08.13".MON_T;
      T     #"AV-08.14".MON_T;
      T     #"AV-08.15".MON_T;
      T     #"AV-08.16".MON_T;
      T     #"AV-08.17".MON_T;
// FB CLOSE Time
      L     t#20s;
      T     #"AV-08.01".MON_T_CLOSE;
      T     #"AV-08.02".MON_T_CLOSE;
      T     #"AV-08.03".MON_T_CLOSE;
      T     #"AV-08.04".MON_T_CLOSE;
      T     #"AV-08.05".MON_T_CLOSE;
      T     #"AV-08.06".MON_T_CLOSE;
      T     #"AV-08.07".MON_T_CLOSE;
      T     #"AV-08.08".MON_T_CLOSE;
      T     #"AV-08.09".MON_T_CLOSE;
      T     #"AV-08.10".MON_T_CLOSE;
      T     #"AV-08.11".MON_T_CLOSE;
      T     #"AV-08.12".MON_T_CLOSE;
      T     #"AV-08.13".MON_T_CLOSE;
      T     #"AV-08.14".MON_T_CLOSE;
      T     #"AV-08.15".MON_T_CLOSE;
      T     #"AV-08.16".MON_T_CLOSE;
      T     #"AV-08.17".MON_T_CLOSE;

REGION Network 3: AV-08.01 w ZSC
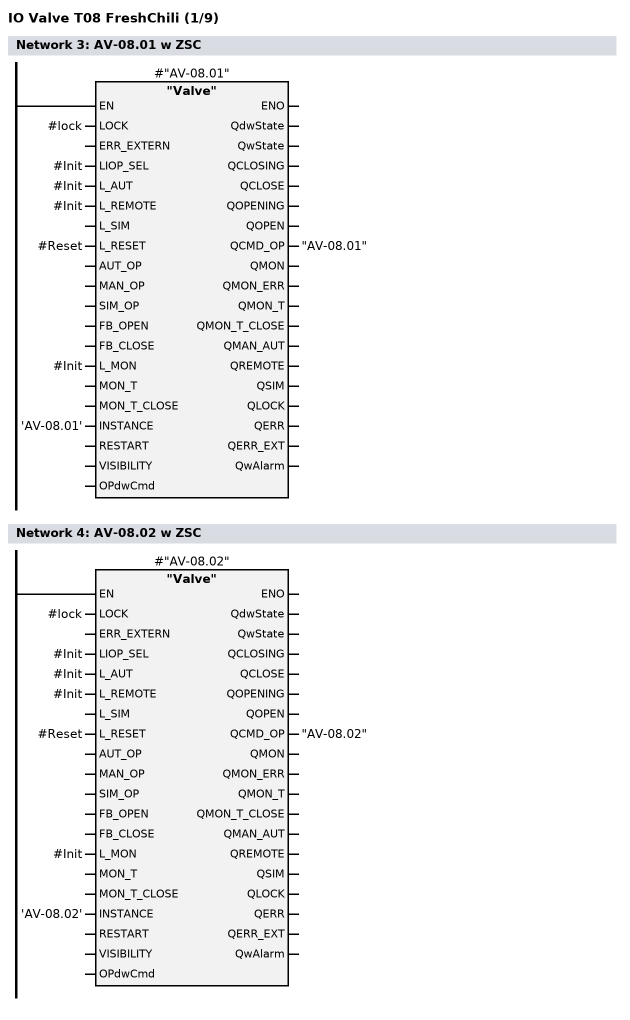
   RUNG wire#powerrail
      #"AV-08.01"(LOCK := #lock, ERR_EXTERN :=, LIOP_SEL := #Init, L_AUT := #Init, L_REMOTE := #Init, L_SIM :=, L_RESET := #Reset, AUT_OP :=, MAN_OP :=, SIM_OP :=, FB_OPEN :=, FB_CLOSE :=, L_MON := #Init, MON_T :=, MON_T_CLOSE :=, INSTANCE := 'AV-08.01', RESTART :=, VISIBILITY :=, OPdwCmd :=, QdwState =>, QwState =>, QCLOSING =>, QCLOSE =>, QOPENING =>, QOPEN =>, QCMD_OP => "AV-08.01", QMON =>, QMON_ERR =>, QMON_T =>, QMON_T_CLOSE =>, QMAN_AUT =>, QREMOTE =>, QSIM =>, QLOCK =>, QERR =>, QERR_EXT =>, QwAlarm =>)
   END_RUNG
   // the same network as SCL:
   #"AV-08.01"(LOCK := #lock,   // "Valve"
               LIOP_SEL := #Init,
               L_AUT := #Init,
               L_REMOTE := #Init,
               L_RESET := #Reset,
               L_MON := #Init,
               INSTANCE := 'AV-08.01',
               QCMD_OP => "AV-08.01");
END_REGION

REGION Network 4: AV-08.02 w ZSC
   RUNG wire#powerrail
      #"AV-08.02"(LOCK := #lock, ERR_EXTERN :=, LIOP_SEL := #Init, L_AUT := #Init, L_REMOTE := #Init, L_SIM :=, L_RESET := #Reset, AUT_OP :=, MAN_OP :=, SIM_OP :=, FB_OPEN :=, FB_CLOSE :=, L_MON := #Init, MON_T :=, MON_T_CLOSE :=, INSTANCE := 'AV-08.02', RESTART :=, VISIBILITY :=, OPdwCmd :=, QdwState =>, QwState =>, QCLOSING =>, QCLOSE =>, QOPENING =>, QOPEN =>, QCMD_OP => "AV-08.02", QMON =>, QMON_ERR =>, QMON_T =>, QMON_T_CLOSE =>, QMAN_AUT =>, QREMOTE =>, QSIM =>, QLOCK =>, QERR =>, QERR_EXT =>, QwAlarm =>)
   END_RUNG
   // the same network as SCL:
   #"AV-08.02"(LOCK := #lock,   // "Valve"
               LIOP_SEL := #Init,
               L_AUT := #Init,
               L_REMOTE := #Init,
               L_RESET := #Reset,
               L_MON := #Init,
               INSTANCE := 'AV-08.02',
               QCMD_OP => "AV-08.02");
END_REGION

REGION Network 5: AV-08.03 w ZSC
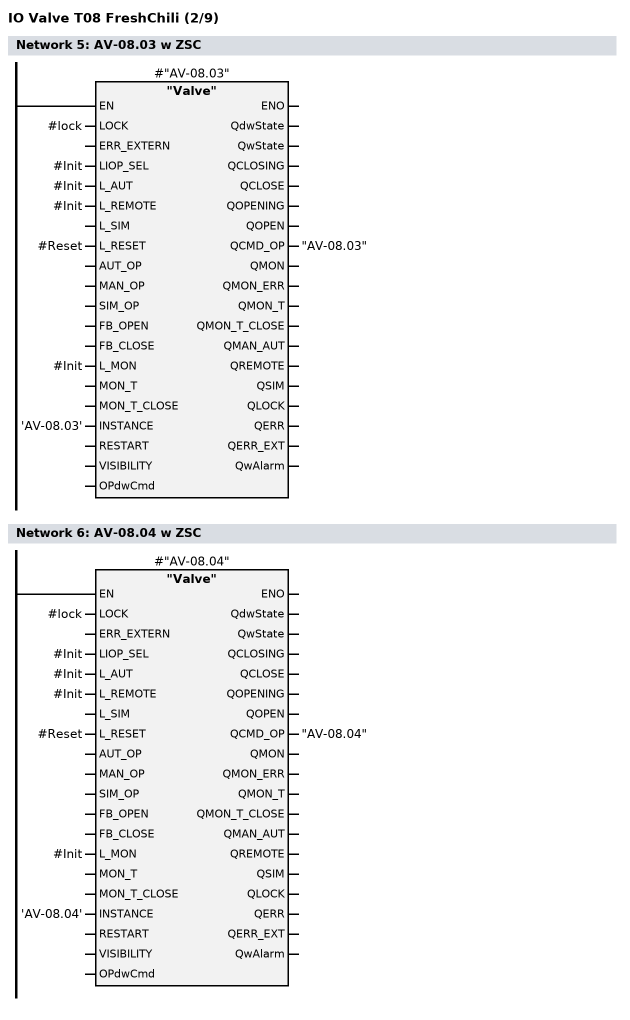
   RUNG wire#powerrail
      #"AV-08.03"(LOCK := #lock, ERR_EXTERN :=, LIOP_SEL := #Init, L_AUT := #Init, L_REMOTE := #Init, L_SIM :=, L_RESET := #Reset, AUT_OP :=, MAN_OP :=, SIM_OP :=, FB_OPEN :=, FB_CLOSE :=, L_MON := #Init, MON_T :=, MON_T_CLOSE :=, INSTANCE := 'AV-08.03', RESTART :=, VISIBILITY :=, OPdwCmd :=, QdwState =>, QwState =>, QCLOSING =>, QCLOSE =>, QOPENING =>, QOPEN =>, QCMD_OP => "AV-08.03", QMON =>, QMON_ERR =>, QMON_T =>, QMON_T_CLOSE =>, QMAN_AUT =>, QREMOTE =>, QSIM =>, QLOCK =>, QERR =>, QERR_EXT =>, QwAlarm =>)
   END_RUNG
   // the same network as SCL:
   #"AV-08.03"(LOCK := #lock,   // "Valve"
               LIOP_SEL := #Init,
               L_AUT := #Init,
               L_REMOTE := #Init,
               L_RESET := #Reset,
               L_MON := #Init,
               INSTANCE := 'AV-08.03',
               QCMD_OP => "AV-08.03");
END_REGION

REGION Network 6: AV-08.04 w ZSC
   RUNG wire#powerrail
      #"AV-08.04"(LOCK := #lock, ERR_EXTERN :=, LIOP_SEL := #Init, L_AUT := #Init, L_REMOTE := #Init, L_SIM :=, L_RESET := #Reset, AUT_OP :=, MAN_OP :=, SIM_OP :=, FB_OPEN :=, FB_CLOSE :=, L_MON := #Init, MON_T :=, MON_T_CLOSE :=, INSTANCE := 'AV-08.04', RESTART :=, VISIBILITY :=, OPdwCmd :=, QdwState =>, QwState =>, QCLOSING =>, QCLOSE =>, QOPENING =>, QOPEN =>, QCMD_OP => "AV-08.04", QMON =>, QMON_ERR =>, QMON_T =>, QMON_T_CLOSE =>, QMAN_AUT =>, QREMOTE =>, QSIM =>, QLOCK =>, QERR =>, QERR_EXT =>, QwAlarm =>)
   END_RUNG
   // the same network as SCL:
   #"AV-08.04"(LOCK := #lock,   // "Valve"
               LIOP_SEL := #Init,
               L_AUT := #Init,
               L_REMOTE := #Init,
               L_RESET := #Reset,
               L_MON := #Init,
               INSTANCE := 'AV-08.04',
               QCMD_OP => "AV-08.04");
END_REGION

REGION Network 7: AV-08.05
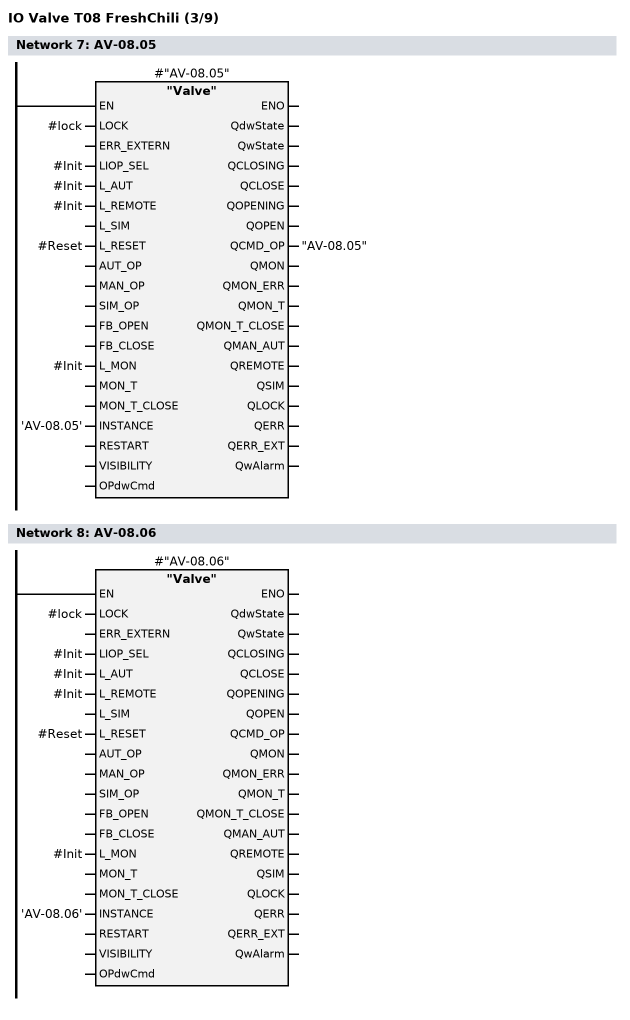
   RUNG wire#powerrail
      #"AV-08.05"(LOCK := #lock, ERR_EXTERN :=, LIOP_SEL := #Init, L_AUT := #Init, L_REMOTE := #Init, L_SIM :=, L_RESET := #Reset, AUT_OP :=, MAN_OP :=, SIM_OP :=, FB_OPEN :=, FB_CLOSE :=, L_MON := #Init, MON_T :=, MON_T_CLOSE :=, INSTANCE := 'AV-08.05', RESTART :=, VISIBILITY :=, OPdwCmd :=, QdwState =>, QwState =>, QCLOSING =>, QCLOSE =>, QOPENING =>, QOPEN =>, QCMD_OP => "AV-08.05", QMON =>, QMON_ERR =>, QMON_T =>, QMON_T_CLOSE =>, QMAN_AUT =>, QREMOTE =>, QSIM =>, QLOCK =>, QERR =>, QERR_EXT =>, QwAlarm =>)
   END_RUNG
   // the same network as SCL:
   #"AV-08.05"(LOCK := #lock,   // "Valve"
               LIOP_SEL := #Init,
               L_AUT := #Init,
               L_REMOTE := #Init,
               L_RESET := #Reset,
               L_MON := #Init,
               INSTANCE := 'AV-08.05',
               QCMD_OP => "AV-08.05");
END_REGION

REGION Network 8: AV-08.06
   RUNG wire#powerrail
      #"AV-08.06"(LOCK := #lock, ERR_EXTERN :=, LIOP_SEL := #Init, L_AUT := #Init, L_REMOTE := #Init, L_SIM :=, L_RESET := #Reset, AUT_OP :=, MAN_OP :=, SIM_OP :=, FB_OPEN :=, FB_CLOSE :=, L_MON := #Init, MON_T :=, MON_T_CLOSE :=, INSTANCE := 'AV-08.06', RESTART :=, VISIBILITY :=, OPdwCmd :=, QdwState =>, QwState =>, QCLOSING =>, QCLOSE =>, QOPENING =>, QOPEN =>, QCMD_OP =>, QMON =>, QMON_ERR =>, QMON_T =>, QMON_T_CLOSE =>, QMAN_AUT =>, QREMOTE =>, QSIM =>, QLOCK =>, QERR =>, QERR_EXT =>, QwAlarm =>)
   END_RUNG
   // the same network as SCL:
   #"AV-08.06"(LOCK := #lock,   // "Valve"
               LIOP_SEL := #Init,
               L_AUT := #Init,
               L_REMOTE := #Init,
               L_RESET := #Reset,
               L_MON := #Init,
               INSTANCE := 'AV-08.06');
END_REGION

REGION Network 9: AV-08.07
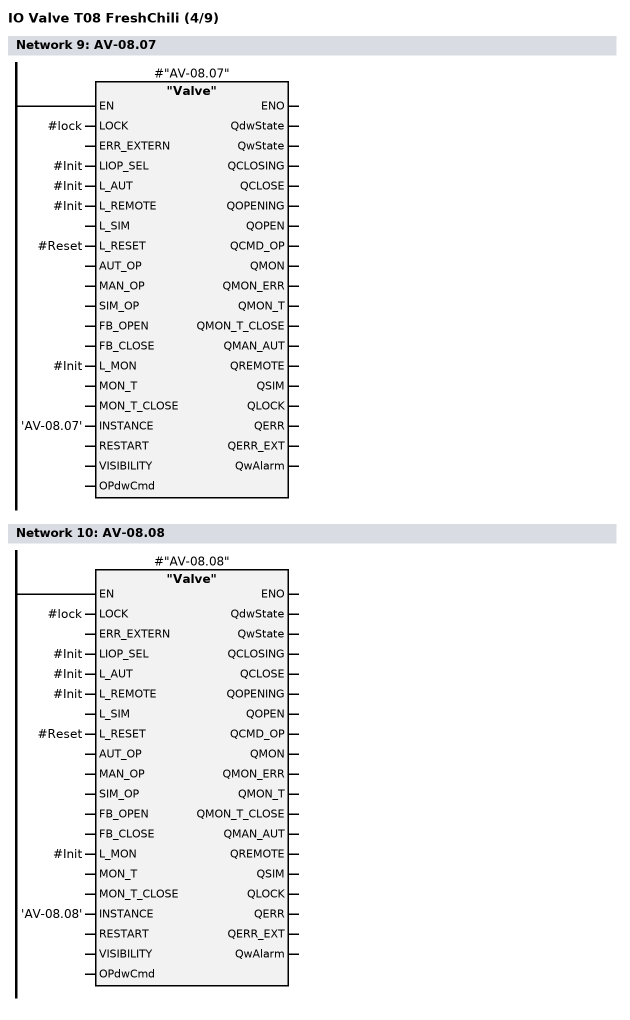
   RUNG wire#powerrail
      #"AV-08.07"(LOCK := #lock, ERR_EXTERN :=, LIOP_SEL := #Init, L_AUT := #Init, L_REMOTE := #Init, L_SIM :=, L_RESET := #Reset, AUT_OP :=, MAN_OP :=, SIM_OP :=, FB_OPEN :=, FB_CLOSE :=, L_MON := #Init, MON_T :=, MON_T_CLOSE :=, INSTANCE := 'AV-08.07', RESTART :=, VISIBILITY :=, OPdwCmd :=, QdwState =>, QwState =>, QCLOSING =>, QCLOSE =>, QOPENING =>, QOPEN =>, QCMD_OP =>, QMON =>, QMON_ERR =>, QMON_T =>, QMON_T_CLOSE =>, QMAN_AUT =>, QREMOTE =>, QSIM =>, QLOCK =>, QERR =>, QERR_EXT =>, QwAlarm =>)
   END_RUNG
   // the same network as SCL:
   #"AV-08.07"(LOCK := #lock,   // "Valve"
               LIOP_SEL := #Init,
               L_AUT := #Init,
               L_REMOTE := #Init,
               L_RESET := #Reset,
               L_MON := #Init,
               INSTANCE := 'AV-08.07');
END_REGION

REGION Network 10: AV-08.08
   RUNG wire#powerrail
      #"AV-08.08"(LOCK := #lock, ERR_EXTERN :=, LIOP_SEL := #Init, L_AUT := #Init, L_REMOTE := #Init, L_SIM :=, L_RESET := #Reset, AUT_OP :=, MAN_OP :=, SIM_OP :=, FB_OPEN :=, FB_CLOSE :=, L_MON := #Init, MON_T :=, MON_T_CLOSE :=, INSTANCE := 'AV-08.08', RESTART :=, VISIBILITY :=, OPdwCmd :=, QdwState =>, QwState =>, QCLOSING =>, QCLOSE =>, QOPENING =>, QOPEN =>, QCMD_OP =>, QMON =>, QMON_ERR =>, QMON_T =>, QMON_T_CLOSE =>, QMAN_AUT =>, QREMOTE =>, QSIM =>, QLOCK =>, QERR =>, QERR_EXT =>, QwAlarm =>)
   END_RUNG
   // the same network as SCL:
   #"AV-08.08"(LOCK := #lock,   // "Valve"
               LIOP_SEL := #Init,
               L_AUT := #Init,
               L_REMOTE := #Init,
               L_RESET := #Reset,
               L_MON := #Init,
               INSTANCE := 'AV-08.08');
END_REGION

REGION Network 11: AV-08.09
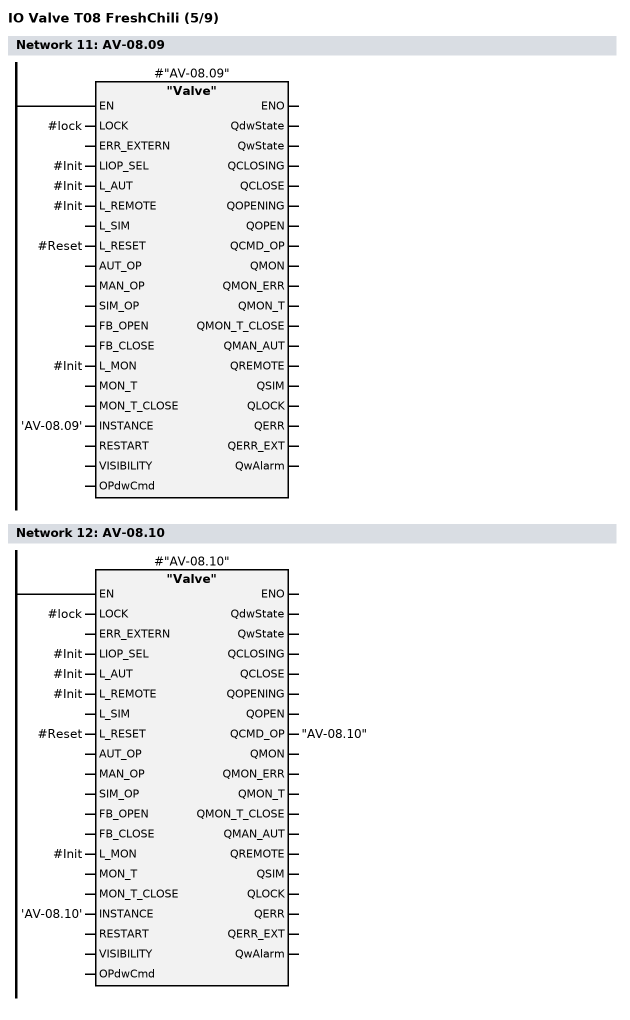
   RUNG wire#powerrail
      #"AV-08.09"(LOCK := #lock, ERR_EXTERN :=, LIOP_SEL := #Init, L_AUT := #Init, L_REMOTE := #Init, L_SIM :=, L_RESET := #Reset, AUT_OP :=, MAN_OP :=, SIM_OP :=, FB_OPEN :=, FB_CLOSE :=, L_MON := #Init, MON_T :=, MON_T_CLOSE :=, INSTANCE := 'AV-08.09', RESTART :=, VISIBILITY :=, OPdwCmd :=, QdwState =>, QwState =>, QCLOSING =>, QCLOSE =>, QOPENING =>, QOPEN =>, QCMD_OP =>, QMON =>, QMON_ERR =>, QMON_T =>, QMON_T_CLOSE =>, QMAN_AUT =>, QREMOTE =>, QSIM =>, QLOCK =>, QERR =>, QERR_EXT =>, QwAlarm =>)
   END_RUNG
   // the same network as SCL:
   #"AV-08.09"(LOCK := #lock,   // "Valve"
               LIOP_SEL := #Init,
               L_AUT := #Init,
               L_REMOTE := #Init,
               L_RESET := #Reset,
               L_MON := #Init,
               INSTANCE := 'AV-08.09');
END_REGION

REGION Network 12: AV-08.10
   RUNG wire#powerrail
      #"AV-08.10"(LOCK := #lock, ERR_EXTERN :=, LIOP_SEL := #Init, L_AUT := #Init, L_REMOTE := #Init, L_SIM :=, L_RESET := #Reset, AUT_OP :=, MAN_OP :=, SIM_OP :=, FB_OPEN :=, FB_CLOSE :=, L_MON := #Init, MON_T :=, MON_T_CLOSE :=, INSTANCE := 'AV-08.10', RESTART :=, VISIBILITY :=, OPdwCmd :=, QdwState =>, QwState =>, QCLOSING =>, QCLOSE =>, QOPENING =>, QOPEN =>, QCMD_OP => "AV-08.10", QMON =>, QMON_ERR =>, QMON_T =>, QMON_T_CLOSE =>, QMAN_AUT =>, QREMOTE =>, QSIM =>, QLOCK =>, QERR =>, QERR_EXT =>, QwAlarm =>)
   END_RUNG
   // the same network as SCL:
   #"AV-08.10"(LOCK := #lock,   // "Valve"
               LIOP_SEL := #Init,
               L_AUT := #Init,
               L_REMOTE := #Init,
               L_RESET := #Reset,
               L_MON := #Init,
               INSTANCE := 'AV-08.10',
               QCMD_OP => "AV-08.10");
END_REGION

REGION Network 13: AV-08.11 w ZSC
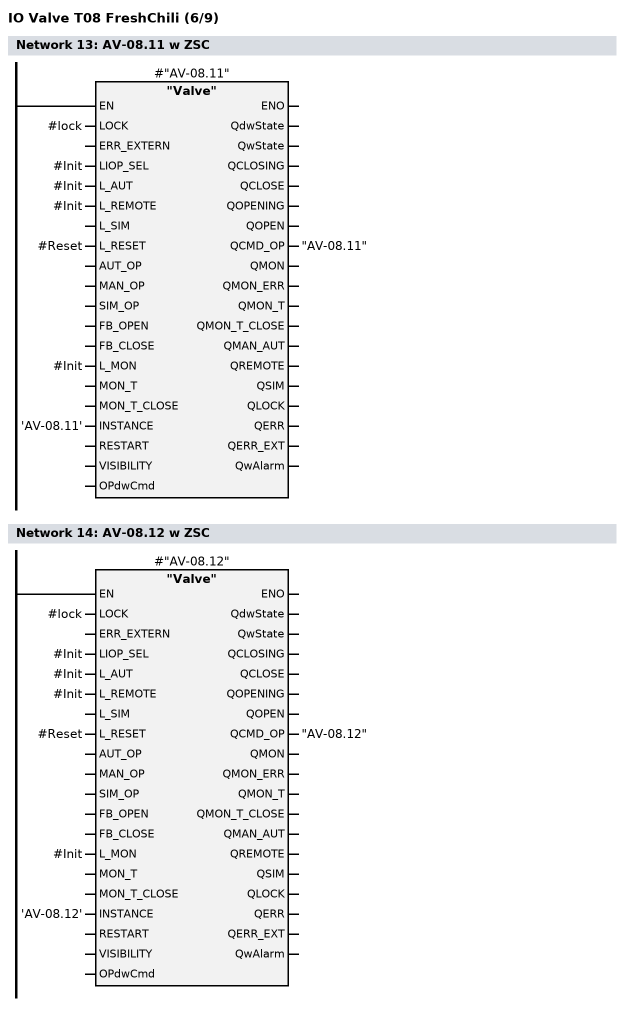
   RUNG wire#powerrail
      #"AV-08.11"(LOCK := #lock, ERR_EXTERN :=, LIOP_SEL := #Init, L_AUT := #Init, L_REMOTE := #Init, L_SIM :=, L_RESET := #Reset, AUT_OP :=, MAN_OP :=, SIM_OP :=, FB_OPEN :=, FB_CLOSE :=, L_MON := #Init, MON_T :=, MON_T_CLOSE :=, INSTANCE := 'AV-08.11', RESTART :=, VISIBILITY :=, OPdwCmd :=, QdwState =>, QwState =>, QCLOSING =>, QCLOSE =>, QOPENING =>, QOPEN =>, QCMD_OP => "AV-08.11", QMON =>, QMON_ERR =>, QMON_T =>, QMON_T_CLOSE =>, QMAN_AUT =>, QREMOTE =>, QSIM =>, QLOCK =>, QERR =>, QERR_EXT =>, QwAlarm =>)
   END_RUNG
   // the same network as SCL:
   #"AV-08.11"(LOCK := #lock,   // "Valve"
               LIOP_SEL := #Init,
               L_AUT := #Init,
               L_REMOTE := #Init,
               L_RESET := #Reset,
               L_MON := #Init,
               INSTANCE := 'AV-08.11',
               QCMD_OP => "AV-08.11");
END_REGION

REGION Network 14: AV-08.12 w ZSC
   RUNG wire#powerrail
      #"AV-08.12"(LOCK := #lock, ERR_EXTERN :=, LIOP_SEL := #Init, L_AUT := #Init, L_REMOTE := #Init, L_SIM :=, L_RESET := #Reset, AUT_OP :=, MAN_OP :=, SIM_OP :=, FB_OPEN :=, FB_CLOSE :=, L_MON := #Init, MON_T :=, MON_T_CLOSE :=, INSTANCE := 'AV-08.12', RESTART :=, VISIBILITY :=, OPdwCmd :=, QdwState =>, QwState =>, QCLOSING =>, QCLOSE =>, QOPENING =>, QOPEN =>, QCMD_OP => "AV-08.12", QMON =>, QMON_ERR =>, QMON_T =>, QMON_T_CLOSE =>, QMAN_AUT =>, QREMOTE =>, QSIM =>, QLOCK =>, QERR =>, QERR_EXT =>, QwAlarm =>)
   END_RUNG
   // the same network as SCL:
   #"AV-08.12"(LOCK := #lock,   // "Valve"
               LIOP_SEL := #Init,
               L_AUT := #Init,
               L_REMOTE := #Init,
               L_RESET := #Reset,
               L_MON := #Init,
               INSTANCE := 'AV-08.12',
               QCMD_OP => "AV-08.12");
END_REGION

REGION Network 15: AV-08.13 w ZSC
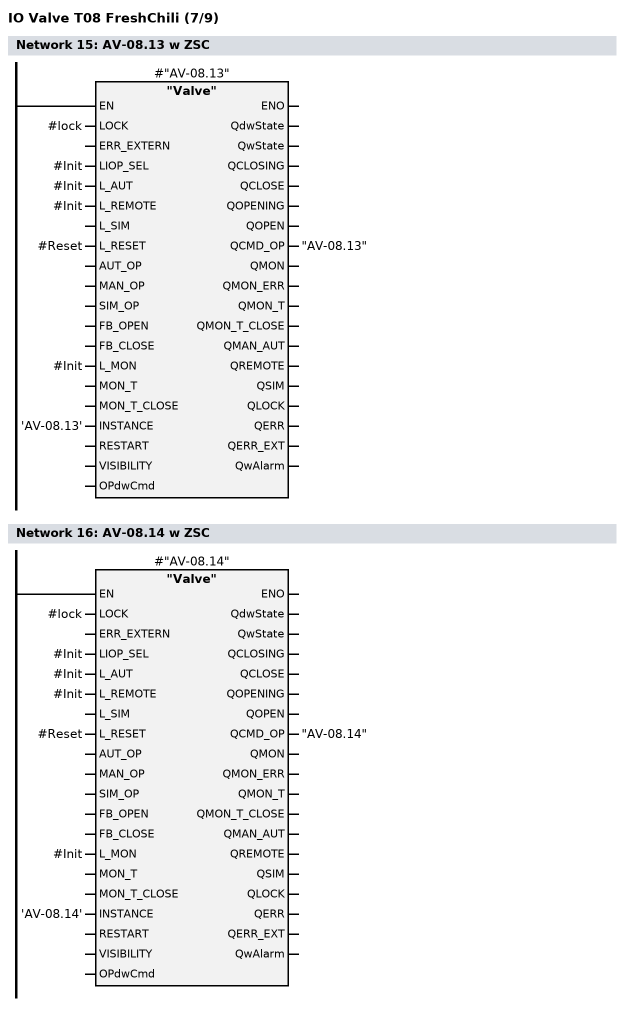
   RUNG wire#powerrail
      #"AV-08.13"(LOCK := #lock, ERR_EXTERN :=, LIOP_SEL := #Init, L_AUT := #Init, L_REMOTE := #Init, L_SIM :=, L_RESET := #Reset, AUT_OP :=, MAN_OP :=, SIM_OP :=, FB_OPEN :=, FB_CLOSE :=, L_MON := #Init, MON_T :=, MON_T_CLOSE :=, INSTANCE := 'AV-08.13', RESTART :=, VISIBILITY :=, OPdwCmd :=, QdwState =>, QwState =>, QCLOSING =>, QCLOSE =>, QOPENING =>, QOPEN =>, QCMD_OP => "AV-08.13", QMON =>, QMON_ERR =>, QMON_T =>, QMON_T_CLOSE =>, QMAN_AUT =>, QREMOTE =>, QSIM =>, QLOCK =>, QERR =>, QERR_EXT =>, QwAlarm =>)
   END_RUNG
   // the same network as SCL:
   #"AV-08.13"(LOCK := #lock,   // "Valve"
               LIOP_SEL := #Init,
               L_AUT := #Init,
               L_REMOTE := #Init,
               L_RESET := #Reset,
               L_MON := #Init,
               INSTANCE := 'AV-08.13',
               QCMD_OP => "AV-08.13");
END_REGION

REGION Network 16: AV-08.14 w ZSC
   RUNG wire#powerrail
      #"AV-08.14"(LOCK := #lock, ERR_EXTERN :=, LIOP_SEL := #Init, L_AUT := #Init, L_REMOTE := #Init, L_SIM :=, L_RESET := #Reset, AUT_OP :=, MAN_OP :=, SIM_OP :=, FB_OPEN :=, FB_CLOSE :=, L_MON := #Init, MON_T :=, MON_T_CLOSE :=, INSTANCE := 'AV-08.14', RESTART :=, VISIBILITY :=, OPdwCmd :=, QdwState =>, QwState =>, QCLOSING =>, QCLOSE =>, QOPENING =>, QOPEN =>, QCMD_OP => "AV-08.14", QMON =>, QMON_ERR =>, QMON_T =>, QMON_T_CLOSE =>, QMAN_AUT =>, QREMOTE =>, QSIM =>, QLOCK =>, QERR =>, QERR_EXT =>, QwAlarm =>)
   END_RUNG
   // the same network as SCL:
   #"AV-08.14"(LOCK := #lock,   // "Valve"
               LIOP_SEL := #Init,
               L_AUT := #Init,
               L_REMOTE := #Init,
               L_RESET := #Reset,
               L_MON := #Init,
               INSTANCE := 'AV-08.14',
               QCMD_OP => "AV-08.14");
END_REGION

REGION Network 17: AV-08.15 w ZSC
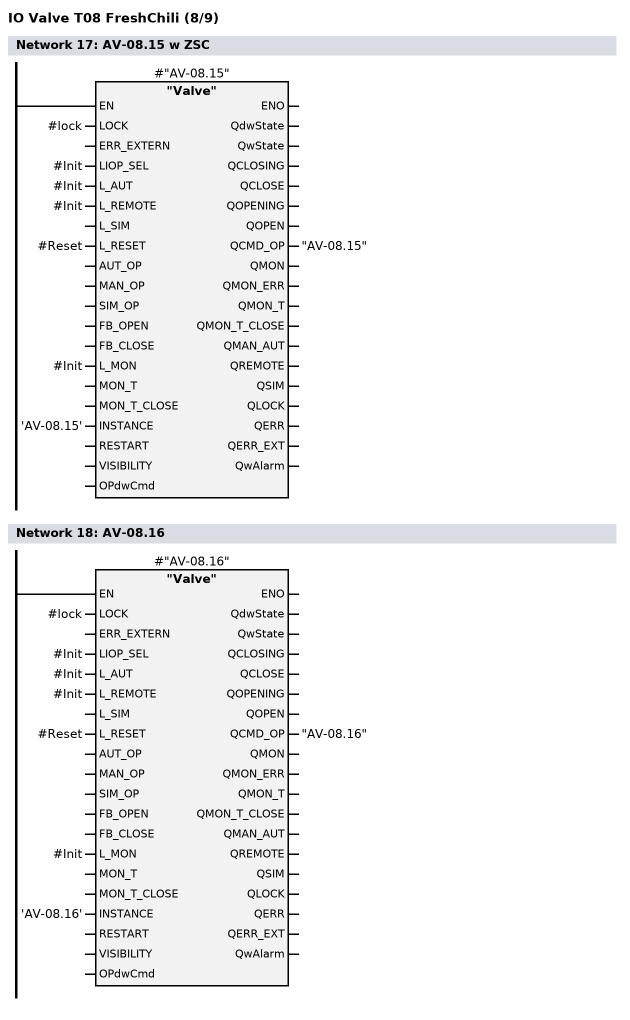
   RUNG wire#powerrail
      #"AV-08.15"(LOCK := #lock, ERR_EXTERN :=, LIOP_SEL := #Init, L_AUT := #Init, L_REMOTE := #Init, L_SIM :=, L_RESET := #Reset, AUT_OP :=, MAN_OP :=, SIM_OP :=, FB_OPEN :=, FB_CLOSE :=, L_MON := #Init, MON_T :=, MON_T_CLOSE :=, INSTANCE := 'AV-08.15', RESTART :=, VISIBILITY :=, OPdwCmd :=, QdwState =>, QwState =>, QCLOSING =>, QCLOSE =>, QOPENING =>, QOPEN =>, QCMD_OP => "AV-08.15", QMON =>, QMON_ERR =>, QMON_T =>, QMON_T_CLOSE =>, QMAN_AUT =>, QREMOTE =>, QSIM =>, QLOCK =>, QERR =>, QERR_EXT =>, QwAlarm =>)
   END_RUNG
   // the same network as SCL:
   #"AV-08.15"(LOCK := #lock,   // "Valve"
               LIOP_SEL := #Init,
               L_AUT := #Init,
               L_REMOTE := #Init,
               L_RESET := #Reset,
               L_MON := #Init,
               INSTANCE := 'AV-08.15',
               QCMD_OP => "AV-08.15");
END_REGION

REGION Network 18: AV-08.16
   RUNG wire#powerrail
      #"AV-08.16"(LOCK := #lock, ERR_EXTERN :=, LIOP_SEL := #Init, L_AUT := #Init, L_REMOTE := #Init, L_SIM :=, L_RESET := #Reset, AUT_OP :=, MAN_OP :=, SIM_OP :=, FB_OPEN :=, FB_CLOSE :=, L_MON := #Init, MON_T :=, MON_T_CLOSE :=, INSTANCE := 'AV-08.16', RESTART :=, VISIBILITY :=, OPdwCmd :=, QdwState =>, QwState =>, QCLOSING =>, QCLOSE =>, QOPENING =>, QOPEN =>, QCMD_OP => "AV-08.16", QMON =>, QMON_ERR =>, QMON_T =>, QMON_T_CLOSE =>, QMAN_AUT =>, QREMOTE =>, QSIM =>, QLOCK =>, QERR =>, QERR_EXT =>, QwAlarm =>)
   END_RUNG
   // the same network as SCL:
   #"AV-08.16"(LOCK := #lock,   // "Valve"
               LIOP_SEL := #Init,
               L_AUT := #Init,
               L_REMOTE := #Init,
               L_RESET := #Reset,
               L_MON := #Init,
               INSTANCE := 'AV-08.16',
               QCMD_OP => "AV-08.16");
END_REGION

REGION Network 19: AV-08.17
